KUKA KRL program: EPS_2_251806_BLK210A_A_20260223023028.src

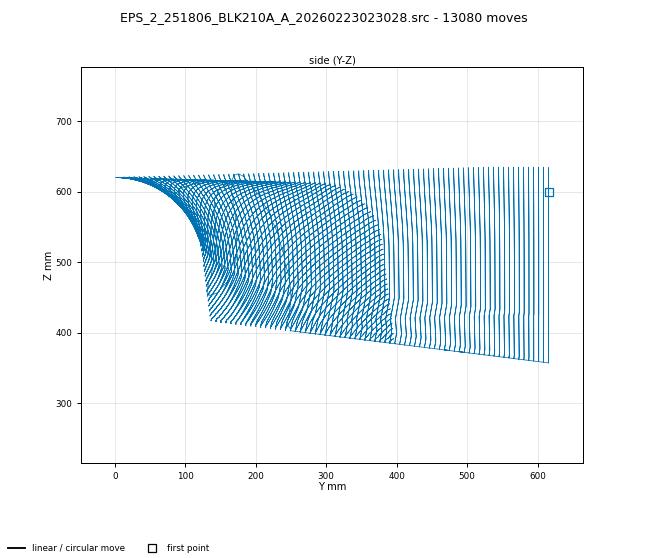
[picture p0: tool path of EPS_2_251806_BLK210A_A_20260223023028.src, 13080 of 13082 moves have a stored position in this frame; points joined in program order, loops and branches not executed]
&ACCESS RVP
&REL 4
&COMMENT QRS 19112012
&PARAM EDITMASK = *
DEF PART()
EXT BAS (BAS_COMMAND :IN,REAL :IN )
INT I
BAS (#INITMOV,0 )

;KUKA QRS Post kuka4.cps  Date:22-06-2017 !

File_ID=3078

QRS_PRE_INIT()

;Init var - Until changes are made in qrs_pre_init
Outlet_Square_prg=0
Inlet_1_Square_prg=0
Inlet_2_Square_prg=0
Inlet_3_Square_prg=0
Inlet_4_Square_prg=0
Inlet_5_Square_prg=0

Outlet_1={X 0.000, Y 530.070, Z 534.500, B 0.000, E1 0.000 }
Inlet_1={X 0.000, Y 550.980, Z 509.500, B 0.000, E1 180.000 }
Outlet_1_type=201
Inlet_1_type=0
;QRS#1=Sidecore dimensions
;QRS#2=200-8" PVC SDR 35
;QRS#3=DeadEnd 201
;QRS#4=
;QRS#5=
;QRS#6=
;QRS#7=
;QRS#8=
;QRS#9=12-08 PSX
;QRS#10=

;QRS#11=
;QRS#12=
;QRS#13=
;QRS#14=
;QRS#15=
;QRS#16=1220x127x914 3'
;QRS#17=EPS Height
;QRS#18=635
;QRS#19=*
;QRS#20= UPDATED VERSION 22-06-2017
;QRS#21=*
Outlet_Square=0100
Inlet_1_Square=00
Inlet_2_Square=0
Inlet_3_Square=0
Inlet_4_Square=0
Inlet_5_Square=0
Mill_Square=1
Outlet_Square_Prg=204
Inlet_1_Square_prg=0

QRS_INIT()

$ADVANCE=5

; T1
PTP {E1 173.602,E2 173.602}
PTP {X 0,Y 615.507,A -85,B 0,C 180,E1 173.602,E2 173.602,E3 0,E4 0,E5 0,E6 0}
QRS_SPEED_INIT()
LIN {X 0,Y 615.507,Z 600,A -85,B 0,C 180,E1 173.602,E2 173.602,E3 0,E4 0,E5 0,E6 0} C_VEL
LIN {X 0,Y 615.507,Z 367.362,A -85,B 0,C 180,E1 173.602,E2 173.602} C_VEL
LIN {X 0,Y 615.507,Z 359.181,A -85,B 0,C 180,E1 173.602,E2 173.602} C_VEL
LIN {X 0,Y 615.49,Z 357.181,A -85,B 0,C 180,E1 173.415,E2 173.415} C_VEL
LIN {X 0,Y 615.478,Z 357.192,A -85,B 0,C 180,E1 170.801,E2 170.801} C_VEL
LIN {X 0,Y 615.484,Z 357.193,A -85,B 0,C 180,E1 168.14,E2 168.14} C_VEL
LIN {X 0,Y 615.49,Z 357.182,A -85,B 0,C 180,E1 165.451,E2 165.451} C_VEL
LIN {X 0,Y 615.489,Z 357.193,A -85,B 0,C 180,E1 162.73,E2 162.73} C_VEL
LIN {X 0,Y 615.483,Z 357.188,A -85,B 0,C 180,E1 159.968,E2 159.968} C_VEL
LIN {X 0,Y 615.491,Z 357.182,A -85,B 0,C 180,E1 157.652,E2 157.652} C_VEL
LIN {X 0,Y 615.477,Z 357.19,A -85,B 0,C 180,E1 155.008,E2 155.008} C_VEL
LIN {X 0,Y 615.482,Z 357.194,A -85,B 0,C 180,E1 152.823,E2 152.823} C_VEL
LIN {X 0,Y 615.482,Z 357.192,A -85,B 0,C 180,E1 150.205,E2 150.205} C_VEL
LIN {X 0,Y 615.489,Z 357.182,A -85,B 0,C 180,E1 147.543,E2 147.543} C_VEL
LIN {X 0,Y 615.477,Z 357.188,A -85,B 0,C 180,E1 145.185,E2 145.185} C_VEL
LIN {X 0,Y 615.491,Z 357.197,A -85,B 0,C 180,E1 142.759,E2 142.759} C_VEL
LIN {X 0,Y 615.487,Z 357.184,A -85,B 0,C 180,E1 139.91,E2 139.91} C_VEL
LIN {X 0,Y 615.493,Z 357.181,A -85,B 0,C 180,E1 137.648,E2 137.648} C_VEL
LIN {X 0,Y 615.481,Z 357.195,A -85,B 0,C 180,E1 134.932,E2 134.932} C_VEL
LIN {X 0,Y 615.482,Z 357.186,A -85,B 0,C 180,E1 132.08,E2 132.08} C_VEL
LIN {X 0,Y 615.494,Z 357.181,A -85,B 0,C 180,E1 129.749,E2 129.749} C_VEL
LIN {X 0,Y 615.483,Z 357.196,A -85,B 0,C 180,E1 126.937,E2 126.937} C_VEL
LIN {X 0,Y 615.492,Z 357.2,A -85,B 0,C 180,E1 124.702,E2 124.702} C_VEL
LIN {X 0,Y 615.48,Z 357.191,A -85,B 0,C 180,E1 122.33,E2 122.33} C_VEL
LIN {X 0,Y 615.497,Z 357.18,A -85,B 0,C 180,E1 119.797,E2 119.797} C_VEL
LIN {X 0,Y 615.486,Z 357.195,A -85,B 0,C 180,E1 117.046,E2 117.046} C_VEL
LIN {X 0,Y 615.479,Z 357.188,A -85,B 0,C 180,E1 114.272,E2 114.272} C_VEL
LIN {X 0,Y 615.477,Z 357.188,A -85,B 0,C 180,E1 111.432,E2 111.432} C_VEL
LIN {X 0,Y 615.482,Z 357.195,A -85,B 0,C 180,E1 108.605,E2 108.605} C_VEL
LIN {X 0,Y 615.486,Z 357.182,A -85,B 0,C 180,E1 105.905,E2 105.905} C_VEL
LIN {X 0,Y 615.48,Z 357.194,A -85,B 0,C 180,E1 103.201,E2 103.201} C_VEL
LIN {X 0,Y 615.479,Z 357.192,A -85,B 0,C 180,E1 100.527,E2 100.527} C_VEL
LIN {X 0,Y 615.488,Z 357.182,A -85,B 0,C 180,E1 97.876,E2 97.876} C_VEL
LIN {X 0,Y 615.482,Z 357.194,A -85,B 0,C 180,E1 95.241,E2 95.241} C_VEL
LIN {X 0,Y 615.477,Z 357.193,A -85,B 0,C 180,E1 92.618,E2 92.618} C_VEL
LIN {X 0,Y 615.486,Z 357.182,A -85,B 0,C 180,E1 90,E2 90} C_VEL
LIN {X 0,Y 615.477,Z 357.193,A -85,B 0,C 180,E1 87.382,E2 87.382} C_VEL
LIN {X 0,Y 615.482,Z 357.194,A -85,B 0,C 180,E1 84.759,E2 84.759} C_VEL
LIN {X 0,Y 615.488,Z 357.182,A -85,B 0,C 180,E1 82.125,E2 82.125} C_VEL
LIN {X 0,Y 615.479,Z 357.192,A -85,B 0,C 180,E1 79.473,E2 79.473} C_VEL
LIN {X 0,Y 615.48,Z 357.194,A -85,B 0,C 180,E1 76.799,E2 76.799} C_VEL
LIN {X 0,Y 615.486,Z 357.182,A -85,B 0,C 180,E1 74.095,E2 74.095} C_VEL
LIN {X 0,Y 615.484,Z 357.196,A -85,B 0,C 180,E1 71.354,E2 71.354} C_VEL
LIN {X 0,Y 615.477,Z 357.188,A -85,B 0,C 180,E1 68.568,E2 68.568} C_VEL
LIN {X 0,Y 615.486,Z 357.183,A -85,B 0,C 180,E1 65.991,E2 65.991} C_VEL
LIN {X 0,Y 615.48,Z 357.192,A -85,B 0,C 180,E1 63.556,E2 63.556} C_VEL
LIN {X 0,Y 615.49,Z 357.197,A -85,B 0,C 180,E1 61.343,E2 61.343} C_VEL
LIN {X 0,Y 615.482,Z 357.193,A -85,B 0,C 180,E1 58.914,E2 58.914} C_VEL
LIN {X 0,Y 615.482,Z 357.184,A -85,B 0,C 180,E1 56.466,E2 56.466} C_VEL
LIN {X 0,Y 615.489,Z 357.182,A -85,B 0,C 180,E1 54.165,E2 54.165} C_VEL
LIN {X 0,Y 615.483,Z 357.185,A -85,B 0,C 180,E1 51.932,E2 51.932} C_VEL
LIN {X 0,Y 615.485,Z 357.2,A -85,B 0,C 180,E1 49.394,E2 49.394} C_VEL
LIN {X 0,Y 615.476,Z 357.189,A -85,B 0,C 180,E1 46.755,E2 46.755} C_VEL
LIN {X 0,Y 615.484,Z 357.185,A -85,B 0,C 180,E1 43.998,E2 43.998} C_VEL
LIN {X 0,Y 615.488,Z 357.198,A -85,B 0,C 180,E1 41.473,E2 41.473} C_VEL
LIN {X 0,Y 615.476,Z 357.191,A -85,B 0,C 180,E1 38.905,E2 38.905} C_VEL
LIN {X 0,Y 615.488,Z 357.182,A -85,B 0,C 180,E1 36.424,E2 36.424} C_VEL
LIN {X 0,Y 615.487,Z 357.198,A -85,B 0,C 180,E1 33.535,E2 33.535} C_VEL
LIN {X 0,Y 615.478,Z 357.189,A -85,B 0,C 180,E1 30.92,E2 30.92} C_VEL
LIN {X 0,Y 615.491,Z 357.181,A -85,B 0,C 180,E1 28.453,E2 28.453} C_VEL
LIN {X 0,Y 615.489,Z 357.198,A -85,B 0,C 180,E1 25.571,E2 25.571} C_VEL
LIN {X 0,Y 615.476,Z 357.187,A -85,B 0,C 180,E1 22.845,E2 22.845} C_VEL
LIN {X 0,Y 615.486,Z 357.182,A -85,B 0,C 180,E1 20.559,E2 20.559} C_VEL
LIN {X 0,Y 615.482,Z 357.19,A -85,B 0,C 180,E1 17.957,E2 17.957} C_VEL
LIN {X 0,Y 615.486,Z 357.192,A -85,B 0,C 180,E1 15.226,E2 15.226} C_VEL
LIN {X 0,Y 615.485,Z 357.183,A -85,B 0,C 180,E1 12.53,E2 12.53} C_VEL
LIN {X 0,Y 615.481,Z 357.194,A -85,B 0,C 180,E1 9.862,E2 9.862} C_VEL
LIN {X 0,Y 615.483,Z 357.191,A -85,B 0,C 180,E1 7.215,E2 7.215} C_VEL
LIN {X 0,Y 615.491,Z 357.181,A -85,B 0,C 180,E1 4.584,E2 4.584} C_VEL
LIN {X 0,Y 615.484,Z 357.192,A -85,B 0,C 180,E1 1.963,E2 1.963} C_VEL
LIN {X 0,Y 615.484,Z 357.193,A -85,B 0,C 180,E1 -0.655,E2 -0.655} C_VEL
LIN {X 0,Y 615.485,Z 357.183,A -85,B 0,C 180,E1 -3.273,E2 -3.273} C_VEL
LIN {X 0,Y 615.484,Z 357.19,A -85,B 0,C 180,E1 -5.899,E2 -5.899} C_VEL
LIN {X 0,Y 615.489,Z 357.194,A -85,B 0,C 180,E1 -8.537,E2 -8.537} C_VEL
LIN {X 0,Y 615.483,Z 357.183,A -85,B 0,C 180,E1 -11.194,E2 -11.194} C_VEL
LIN {X 0,Y 615.485,Z 357.192,A -85,B 0,C 180,E1 -13.935,E2 -13.935} C_VEL
LIN {X 0,Y 615.481,Z 357.192,A -85,B 0,C 180,E1 -16.587,E2 -16.587} C_VEL
LIN {X 0,Y 615.486,Z 357.183,A -85,B 0,C 180,E1 -19.338,E2 -19.338} C_VEL
LIN {X 0,Y 615.493,Z 357.2,A -85,B 0,C 180,E1 -22.137,E2 -22.137} C_VEL
LIN {X 0,Y 615.476,Z 357.185,A -85,B 0,C 180,E1 -24.993,E2 -24.993} C_VEL
LIN {X 0,Y 615.481,Z 357.184,A -85,B 0,C 180,E1 -27.178,E2 -27.178} C_VEL
LIN {X 0,Y 615.485,Z 357.192,A -85,B 0,C 180,E1 -29.796,E2 -29.796} C_VEL
LIN {X 0,Y 615.489,Z 357.191,A -85,B 0,C 180,E1 -32.458,E2 -32.458} C_VEL
LIN {X 0,Y 615.477,Z 357.186,A -85,B 0,C 180,E1 -34.816,E2 -34.816} C_VEL
LIN {X 0,Y 615.489,Z 357.182,A -85,B 0,C 180,E1 -37.242,E2 -37.242} C_VEL
LIN {X 0,Y 615.498,Z 357.2,A -85,B 0,C 180,E1 -40.091,E2 -40.091} C_VEL
LIN {X 0,Y 615.493,Z 357.191,A -85,B 0,C 180,E1 -42.353,E2 -42.353} C_VEL
LIN {X 0,Y 615.481,Z 357.184,A -85,B 0,C 180,E1 -45.07,E2 -45.07} C_VEL
LIN {X 0,Y 615.489,Z 357.199,A -85,B 0,C 180,E1 -47.92,E2 -47.92} C_VEL
LIN {X 0,Y 615.495,Z 357.192,A -85,B 0,C 180,E1 -50.251,E2 -50.251} C_VEL
LIN {X 0,Y 615.483,Z 357.183,A -85,B 0,C 180,E1 -53.064,E2 -53.064} C_VEL
LIN {X 0,Y 615.496,Z 357.2,A -85,B 0,C 180,E1 -55.979,E2 -55.979} C_VEL
LIN {X 0,Y 615.482,Z 357.183,A -85,B 0,C 180,E1 -58.915,E2 -58.915} C_VEL
LIN {X 0,Y 615.486,Z 357.191,A -85,B 0,C 180,E1 -61.551,E2 -61.551} C_VEL
LIN {X 0,Y 615.481,Z 357.188,A -85,B 0,C 180,E1 -64.433,E2 -64.433} C_VEL
LIN {X 0,Y 615.497,Z 357.361,A -85,B 0,C 180,E1 -65.958,E2 -65.958} C_VEL
LIN {X 0,Y 615.496,Z 372.441,A -85,B 0,C 180,E1 -68.569,E2 -68.569} C_VEL
LIN {X 0,Y 615.482,Z 389.222,A -85,B 0,C 180,E1 -71.398,E2 -71.398} C_VEL
LIN {X 0,Y 615.49,Z 405.467,A -85,B 0,C 180,E1 -74.095,E2 -74.095} C_VEL
LIN {X 0,Y 615.497,Z 422.987,A -85,B 0,C 180,E1 -76.967,E2 -76.967} C_VEL
LIN {X 0,Y 615.495,Z 424.551,A -85,B 0,C 180,E1 -77.135,E2 -77.135} C_VEL
LIN {X 0,Y 615.497,Z 530.847,A -85,B 0,C 180,E1 -78.411,E2 -78.411} C_VEL
LIN {X 0,Y 615.499,Z 543.354,A -85,B 0,C 180,E1 -78.682,E2 -78.682} C_VEL
LIN {X 0,Y 615.496,Z 556.502,A -85,B 0,C 180,E1 -79.109,E2 -79.109} C_VEL
LIN {X 0,Y 615.484,Z 568.484,A -85,B 0,C 180,E1 -79.64,E2 -79.64} C_VEL
LIN {X 0,Y 615.487,Z 580,A -85,B 0,C 180,E1 -80.304,E2 -80.304} C_VEL
LIN {X 0,Y 615.499,Z 590.345,A -85,B 0,C 180,E1 -81.05,E2 -81.05} C_VEL
LIN {X 0,Y 615.497,Z 598.815,A -85,B 0,C 180,E1 -81.794,E2 -81.794} C_VEL
LIN {X 0,Y 615.498,Z 606.609,A -85,B 0,C 180,E1 -82.62,E2 -82.62} C_VEL
LIN {X 0,Y 615.496,Z 614.205,A -85,B 0,C 180,E1 -83.608,E2 -83.608} C_VEL
LIN {X 0,Y 615.498,Z 621.206,A -85,B 0,C 180,E1 -84.759,E2 -84.759} C_VEL
LIN {X 0,Y 615.493,Z 625.853,A -85,B 0,C 180,E1 -85.744,E2 -85.744} C_VEL
LIN {X 0,Y 615.495,Z 629.399,A -85,B 0,C 180,E1 -86.727,E2 -86.727} C_VEL
LIN {X 0,Y 615.497,Z 631.233,A -85,B 0,C 180,E1 -87.382,E2 -87.382} C_VEL
LIN {X 0,Y 615.497,Z 632.608,A -85,B 0,C 180,E1 -88.037,E2 -88.037} C_VEL
LIN {X 0,Y 615.496,Z 634.174,A -85,B 0,C 180,E1 -89.346,E2 -89.346} C_VEL
LIN {X 0,Y 615.494,Z 634.389,A -85,B 0,C 180,E1 -90,E2 -90} C_VEL
LIN {X 0,Y 615.496,Z 633.58,A -85,B 0,C 180,E1 -91.309,E2 -91.309} C_VEL
LIN {X 0,Y 615.497,Z 632.608,A -85,B 0,C 180,E1 -91.963,E2 -91.963} C_VEL
LIN {X 0,Y 615.497,Z 631.232,A -85,B 0,C 180,E1 -92.618,E2 -92.618} C_VEL
LIN {X 0,Y 615.496,Z 628.349,A -85,B 0,C 180,E1 -93.601,E2 -93.601} C_VEL
LIN {X 0,Y 615.498,Z 624.441,A -85,B 0,C 180,E1 -94.585,E2 -94.585} C_VEL
LIN {X 0,Y 615.499,Z 619.404,A -85,B 0,C 180,E1 -95.57,E2 -95.57} C_VEL
LIN {X 0,Y 615.497,Z 612.87,A -85,B 0,C 180,E1 -96.583,E2 -96.583} C_VEL
LIN {X 0,Y 615.497,Z 605.132,A -85,B 0,C 180,E1 -97.545,E2 -97.545} C_VEL
LIN {X 0,Y 615.498,Z 597.044,A -85,B 0,C 180,E1 -98.371,E2 -98.371} C_VEL
LIN {X 0,Y 615.499,Z 587.166,A -85,B 0,C 180,E1 -99.199,E2 -99.199} C_VEL
LIN {X 0,Y 615.488,Z 575.98,A -85,B 0,C 180,E1 -99.945,E2 -99.945} C_VEL
LIN {X 0,Y 615.486,Z 565.021,A -85,B 0,C 180,E1 -100.527,E2 -100.527} C_VEL
LIN {X 0,Y 615.499,Z 552.418,A -85,B 0,C 180,E1 -101.042,E2 -101.042} C_VEL
LIN {X 0,Y 615.499,Z 540.06,A -85,B 0,C 180,E1 -101.401,E2 -101.401} C_VEL
LIN {X 0,Y 615.498,Z 526.459,A -85,B 0,C 180,E1 -101.652,E2 -101.652} C_VEL
LIN {X 0,Y 615.495,Z 424.541,A -85,B 0,C 180,E1 -102.865,E2 -102.865} C_VEL
LIN {X 0,Y 615.497,Z 422.984,A -85,B 0,C 180,E1 -103.033,E2 -103.033} C_VEL
LIN {X 0,Y 615.49,Z 405.464,A -85,B 0,C 180,E1 -105.905,E2 -105.905} C_VEL
LIN {X 0,Y 615.484,Z 388.96,A -85,B 0,C 180,E1 -108.646,E2 -108.646} C_VEL
LIN {X 0,Y 615.496,Z 372.438,A -85,B 0,C 180,E1 -111.432,E2 -111.432} C_VEL
LIN {X 0,Y 615.497,Z 357.361,A -85,B 0,C 180,E1 -114.042,E2 -114.042} C_VEL
LIN {X 0,Y 615.485,Z 357.192,A -85,B 0,C 180,E1 -116.444,E2 -116.444} C_VEL
LIN {X 0,Y 615.489,Z 357.186,A -85,B 0,C 180,E1 -118.658,E2 -118.658} C_VEL
LIN {X 0,Y 615.482,Z 357.183,A -85,B 0,C 180,E1 -121.085,E2 -121.085} C_VEL
LIN {X 0,Y 615.498,Z 357.199,A -85,B 0,C 180,E1 -124.021,E2 -124.021} C_VEL
LIN {X 0,Y 615.483,Z 357.183,A -85,B 0,C 180,E1 -126.936,E2 -126.936} C_VEL
LIN {X 0,Y 615.495,Z 357.192,A -85,B 0,C 180,E1 -129.749,E2 -129.749} C_VEL
LIN {X 0,Y 615.485,Z 357.191,A -85,B 0,C 180,E1 -132.353,E2 -132.353} C_VEL
LIN {X 0,Y 615.479,Z 357.184,A -85,B 0,C 180,E1 -135.069,E2 -135.069} C_VEL
LIN {X 0,Y 615.496,Z 357.2,A -85,B 0,C 180,E1 -137.918,E2 -137.918} C_VEL
LIN {X 0,Y 615.486,Z 357.192,A -85,B 0,C 180,E1 -140.249,E2 -140.249} C_VEL
LIN {X 0,Y 615.478,Z 357.185,A -85,B 0,C 180,E1 -143.064,E2 -143.064} C_VEL
LIN {X 0,Y 615.495,Z 357.198,A -85,B 0,C 180,E1 -145.978,E2 -145.978} C_VEL
LIN {X 0,Y 615.485,Z 357.189,A -85,B 0,C 180,E1 -148.314,E2 -148.314} C_VEL
LIN {X 0,Y 615.488,Z 357.183,A -85,B 0,C 180,E1 -150.593,E2 -150.593} C_VEL
LIN {X 0,Y 615.481,Z 357.184,A -85,B 0,C 180,E1 -152.955,E2 -152.955} C_VEL
LIN {X 0,Y 615.496,Z 357.197,A -85,B 0,C 180,E1 -155.728,E2 -155.728} C_VEL
LIN {X 0,Y 615.495,Z 357.182,A -85,B 0,C 180,E1 -158.568,E2 -158.568} C_VEL
LIN {X 0,Y 615.485,Z 357.191,A -85,B 0,C 180,E1 -161.395,E2 -161.395} C_VEL
LIN {X 0,Y 615.483,Z 357.193,A -85,B 0,C 180,E1 -164.094,E2 -164.094} C_VEL
LIN {X 0,Y 615.484,Z 357.183,A -85,B 0,C 180,E1 -166.798,E2 -166.798} C_VEL
LIN {X 0,Y 615.493,Z 357.193,A -85,B 0,C 180,E1 -169.473,E2 -169.473} C_VEL
LIN {X 0,Y 615.482,Z 357.19,A -85,B 0,C 180,E1 -172.124,E2 -172.124} C_VEL
LIN {X 0,Y 615.484,Z 357.183,A -85,B 0,C 180,E1 -174.758,E2 -174.758} C_VEL
LIN {X 0,Y 615.489,Z 357.192,A -85,B 0,C 180,E1 -177.382,E2 -177.382} C_VEL
LIN {X 0,Y 615.484,Z 357.192,A -85,B 0,C 180,E1 -180,E2 -180} C_VEL
LIN {X 0,Y 615.49,Z 357.182,A -85,B 0,C 180,E1 -182.617,E2 -182.617} C_VEL
LIN {X 0,Y 615.484,Z 357.191,A -85,B 0,C 180,E1 -185.241,E2 -185.241} C_VEL
LIN {X 0,Y 615.49,Z 357.181,A -85,B 0,C 180,E1 -186.585,E2 -186.585} C_VEL
LIN {X 0,Y 614.809,Z 357.338,A -85,B 0,C 180,E1 -187.131,E2 -187.131} C_VEL
LIN {X 0,Y 611.968,Z 357.753,A -85,B 0,C 180,E1 -188.017,E2 -188.017} C_VEL
LIN {X 0,Y 609.575,Z 358.065,A -85,B 0,C 180,E1 -188.729,E2 -188.729} C_VEL
LIN {X 0,Y 608.541,Z 358.183,A -85,B 0,C 180,E1 -189.279,E2 -189.279} C_VEL
LIN {X 0,Y 608.453,Z 358.191,A -85,B 0,C 180,E1 -189.465,E2 -189.465} C_VEL
LIN {X 0,Y 608.46,Z 358.19,A -85,B 0,C 180,E1 -191.999,E2 -191.999} C_VEL
LIN {X 0,Y 608.477,Z 358.185,A -85,B 0,C 180,E1 -194.72,E2 -194.72} C_VEL
LIN {X 0,Y 608.453,Z 358.197,A -85,B 0,C 180,E1 -197.476,E2 -197.476} C_VEL
LIN {X 0,Y 608.461,Z 358.186,A -85,B 0,C 180,E1 -200.274,E2 -200.274} C_VEL
LIN {X 0,Y 608.455,Z 358.187,A -85,B 0,C 180,E1 -202.476,E2 -202.476} C_VEL
LIN {X 0,Y 608.451,Z 358.187,A -85,B 0,C 180,E1 -204.571,E2 -204.571} C_VEL
LIN {X 0,Y 608.474,Z 358.191,A -85,B 0,C 180,E1 -207.207,E2 -207.207} C_VEL
LIN {X 0,Y 608.465,Z 358.188,A -85,B 0,C 180,E1 -209.972,E2 -209.972} C_VEL
LIN {X 0,Y 608.463,Z 358.186,A -85,B 0,C 180,E1 -212.523,E2 -212.523} C_VEL
LIN {X 0,Y 608.44,Z 358.197,A -85,B 0,C 180,E1 -215.277,E2 -215.277} C_VEL
LIN {X 0,Y 608.469,Z 358.19,A -85,B 0,C 180,E1 -217.746,E2 -217.746} C_VEL
LIN {X 0,Y 608.449,Z 358.187,A -85,B 0,C 180,E1 -220.329,E2 -220.329} C_VEL
LIN {X 0,Y 608.483,Z 358.194,A -85,B 0,C 180,E1 -223.311,E2 -223.311} C_VEL
LIN {X 0,Y 608.468,Z 358.185,A -85,B 0,C 180,E1 -226.131,E2 -226.131} C_VEL
LIN {X 0,Y 608.449,Z 358.19,A -85,B 0,C 180,E1 -228.823,E2 -228.823} C_VEL
LIN {X 0,Y 608.468,Z 358.194,A -85,B 0,C 180,E1 -231.412,E2 -231.412} C_VEL
LIN {X 0,Y 608.475,Z 358.185,A -85,B 0,C 180,E1 -233.95,E2 -233.95} C_VEL
LIN {X 0,Y 608.46,Z 358.186,A -85,B 0,C 180,E1 -236.329,E2 -236.329} C_VEL
LIN {X 0,Y 608.474,Z 358.187,A -85,B 0,C 180,E1 -238.727,E2 -238.727} C_VEL
LIN {X 0,Y 608.473,Z 358.192,A -85,B 0,C 180,E1 -241.379,E2 -241.379} C_VEL
LIN {X 0,Y 608.47,Z 358.185,A -85,B 0,C 180,E1 -244.278,E2 -244.278} C_VEL
LIN {X 0,Y 608.449,Z 358.193,A -85,B 0,C 180,E1 -246.876,E2 -246.876} C_VEL
LIN {X 0,Y 608.46,Z 358.188,A -85,B 0,C 180,E1 -249.726,E2 -249.726} C_VEL
LIN {X 0,Y 608.45,Z 358.189,A -85,B 0,C 180,E1 -252.523,E2 -252.523} C_VEL
LIN {X 0,Y 608.469,Z 358.193,A -85,B 0,C 180,E1 -255.279,E2 -255.279} C_VEL
LIN {X 0,Y 608.461,Z 358.186,A -85,B 0,C 180,E1 -258,E2 -258} C_VEL
LIN {X 0,Y 608.466,Z 358.19,A -85,B 0,C 180,E1 -260.694,E2 -260.694} C_VEL
LIN {X 0,Y 608.475,Z 358.19,A -85,B 0,C 180,E1 -263.367,E2 -263.367} C_VEL
LIN {X 0,Y 608.455,Z 358.187,A -85,B 0,C 180,E1 -266.026,E2 -266.026} C_VEL
LIN {X 0,Y 608.465,Z 358.191,A -85,B 0,C 180,E1 -268.676,E2 -268.676} C_VEL
LIN {X 0,Y 608.465,Z 358.191,A -85,B 0,C 180,E1 -271.323,E2 -271.323} C_VEL
LIN {X 0,Y 608.456,Z 358.187,A -85,B 0,C 180,E1 -273.974,E2 -273.974} C_VEL
LIN {X 0,Y 608.474,Z 358.19,A -85,B 0,C 180,E1 -276.632,E2 -276.632} C_VEL
LIN {X 0,Y 608.466,Z 358.19,A -85,B 0,C 180,E1 -279.306,E2 -279.306} C_VEL
LIN {X 0,Y 608.461,Z 358.186,A -85,B 0,C 180,E1 -281.999,E2 -281.999} C_VEL
LIN {X 0,Y 608.469,Z 358.193,A -85,B 0,C 180,E1 -284.72,E2 -284.72} C_VEL
LIN {X 0,Y 608.45,Z 358.189,A -85,B 0,C 180,E1 -287.476,E2 -287.476} C_VEL
LIN {X 0,Y 608.46,Z 358.188,A -85,B 0,C 180,E1 -290.274,E2 -290.274} C_VEL
LIN {X 0,Y 608.449,Z 358.193,A -85,B 0,C 180,E1 -293.124,E2 -293.124} C_VEL
LIN {X 0,Y 608.47,Z 358.185,A -85,B 0,C 180,E1 -295.722,E2 -295.722} C_VEL
LIN {X 0,Y 608.472,Z 358.192,A -85,B 0,C 180,E1 -298.621,E2 -298.621} C_VEL
LIN {X 0,Y 608.472,Z 358.187,A -85,B 0,C 180,E1 -301.316,E2 -301.316} C_VEL
LIN {X 0,Y 608.469,Z 358.185,A -85,B 0,C 180,E1 -303.735,E2 -303.735} C_VEL
LIN {X 0,Y 608.473,Z 358.186,A -85,B 0,C 180,E1 -306.09,E2 -306.09} C_VEL
LIN {X 0,Y 608.468,Z 358.194,A -85,B 0,C 180,E1 -308.587,E2 -308.587} C_VEL
LIN {X 0,Y 608.456,Z 358.187,A -85,B 0,C 180,E1 -311.342,E2 -311.342} C_VEL
LIN {X 0,Y 608.45,Z 358.191,A -85,B 0,C 180,E1 -314.264,E2 -314.264} C_VEL
LIN {X 0,Y 608.452,Z 358.192,A -85,B 0,C 180,E1 -317.041,E2 -317.041} C_VEL
LIN {X 0,Y 608.45,Z 358.187,A -85,B 0,C 180,E1 -319.697,E2 -319.697} C_VEL
LIN {X 0,Y 608.469,Z 358.19,A -85,B 0,C 180,E1 -322.254,E2 -322.254} C_VEL
LIN {X 0,Y 608.469,Z 358.188,A -85,B 0,C 180,E1 -325.09,E2 -325.09} C_VEL
LIN {X 0,Y 608.471,Z 358.186,A -85,B 0,C 180,E1 -327.906,E2 -327.906} C_VEL
LIN {X 0,Y 608.467,Z 358.19,A -85,B 0,C 180,E1 -330.221,E2 -330.221} C_VEL
LIN {X 0,Y 608.474,Z 358.191,A -85,B 0,C 180,E1 -332.792,E2 -332.792} C_VEL
LIN {X 0,Y 608.451,Z 358.187,A -85,B 0,C 180,E1 -335.429,E2 -335.429} C_VEL
LIN {X 0,Y 608.475,Z 358.192,A -85,B 0,C 180,E1 -338.309,E2 -338.309} C_VEL
LIN {X 0,Y 608.466,Z 358.186,A -85,B 0,C 180,E1 -341.283,E2 -341.283} C_VEL
LIN {X 0,Y 608.46,Z 358.188,A -85,B 0,C 180,E1 -343.907,E2 -343.907} C_VEL
LIN {X 0,Y 608.461,Z 358.193,A -85,B 0,C 180,E1 -346.644,E2 -346.644} C_VEL
LIN {X 0,Y 608.465,Z 358.185,A -85,B 0,C 180,E1 -349.351,E2 -349.351} C_VEL
LIN {X 0,Y 608.476,Z 358.188,A -85,B 0,C 180,E1 -352.033,E2 -352.033} C_VEL
LIN {X 0,Y 608.463,Z 358.191,A -85,B 0,C 180,E1 -354.699,E2 -354.699} C_VEL
LIN {X 0,Y 608.48,Z 358.184,A -85,B 0,C 180,E1 -357.352,E2 -357.352} C_VEL
LIN {X 0,Y 608.472,Z 358.189,A -85,B 0,C 180,E1 -360,E2 -360} C_VEL
LIN {X 0,Y 608.48,Z 358.189,A -85,B 0,C 180,E1 -362.648,E2 -362.648} C_VEL
LIN {X 0,Y 608.463,Z 358.186,A -85,B 0,C 180,E1 -365.302,E2 -365.302} C_VEL
LIN {X 0,Y 608.474,Z 358.189,A -85,B 0,C 180,E1 -367.967,E2 -367.967} C_VEL
LIN {X 0,Y 608.463,Z 358.187,A -85,B 0,C 180,E1 -370.957,E2 -370.957} C_VEL
LIN {X 0,Y 608.461,Z 358.186,A -85,B 0,C 180,E1 -373.357,E2 -373.357} C_VEL
LIN {X 0,Y 608.46,Z 358.194,A -85,B 0,C 180,E1 -376.094,E2 -376.094} C_VEL
LIN {X 0,Y 608.452,Z 358.188,A -85,B 0,C 180,E1 -378.87,E2 -378.87} C_VEL
LIN {X 0,Y 608.476,Z 358.187,A -85,B 0,C 180,E1 -381.692,E2 -381.692} C_VEL
LIN {X 0,Y 608.452,Z 358.191,A -85,B 0,C 180,E1 -384.571,E2 -384.571} C_VEL
LIN {X 0,Y 608.473,Z 358.184,A -85,B 0,C 180,E1 -387.208,E2 -387.208} C_VEL
LIN {X 0,Y 608.47,Z 358.193,A -85,B 0,C 180,E1 -389.974,E2 -389.974} C_VEL
LIN {X 0,Y 608.463,Z 358.19,A -85,B 0,C 180,E1 -392.524,E2 -392.524} C_VEL
LIN {X 0,Y 608.439,Z 358.189,A -85,B 0,C 180,E1 -395.278,E2 -395.278} C_VEL
LIN {X 0,Y 608.473,Z 358.19,A -85,B 0,C 180,E1 -397.746,E2 -397.746} C_VEL
LIN {X 0,Y 608.454,Z 358.193,A -85,B 0,C 180,E1 -400.33,E2 -400.33} C_VEL
LIN {X 0,Y 608.453,Z 358.187,A -85,B 0,C 180,E1 -402.96,E2 -402.96} C_VEL
LIN {X 0,Y 608.457,Z 358.192,A -85,B 0,C 180,E1 -405.736,E2 -405.736} C_VEL
LIN {X 0,Y 608.457,Z 358.188,A -85,B 0,C 180,E1 -408.659,E2 -408.659} C_VEL
LIN {X 0,Y 608.471,Z 358.187,A -85,B 0,C 180,E1 -411.413,E2 -411.413} C_VEL
LIN {X 0,Y 608.479,Z 358.195,A -85,B 0,C 180,E1 -413.951,E2 -413.951} C_VEL
LIN {X 0,Y 608.464,Z 358.19,A -85,B 0,C 180,E1 -416.33,E2 -416.33} C_VEL
LIN {X 0,Y 608.46,Z 358.187,A -85,B 0,C 180,E1 -418.731,E2 -418.731} C_VEL
LIN {X 0,Y 608.474,Z 358.187,A -85,B 0,C 180,E1 -421.38,E2 -421.38} C_VEL
LIN {X 0,Y 608.471,Z 358.19,A -85,B 0,C 180,E1 -424.28,E2 -424.28} C_VEL
LIN {X 0,Y 608.491,Z 358.355,A -85,B 0,C 180,E1 -425.845,E2 -425.845} C_VEL
LIN {X 0,Y 608.547,Z 372.465,A -85,B 0,C 180,E1 -428.312,E2 -428.312} C_VEL
LIN {X 0,Y 608.511,Z 389.856,A -85,B 0,C 180,E1 -431.274,E2 -431.274} C_VEL
LIN {X 0,Y 608.496,Z 406.613,A -85,B 0,C 180,E1 -434.08,E2 -434.08} C_VEL
LIN {X 0,Y 608.473,Z 424.032,A -85,B 0,C 180,E1 -436.942,E2 -436.942} C_VEL
LIN {X 0,Y 608.582,Z 425.271,A -85,B 0,C 180,E1 -437.008,E2 -437.008} C_VEL
LIN {X 0,Y 608.549,Z 530.958,A -85,B 0,C 180,E1 -438.277,E2 -438.277} C_VEL
LIN {X 0,Y 608.547,Z 544.234,A -85,B 0,C 180,E1 -438.572,E2 -438.572} C_VEL
LIN {X 0,Y 608.54,Z 557.395,A -85,B 0,C 180,E1 -439.011,E2 -439.011} C_VEL
LIN {X 0,Y 608.507,Z 568.632,A -85,B 0,C 180,E1 -439.52,E2 -439.52} C_VEL
LIN {X 0,Y 608.48,Z 580.198,A -85,B 0,C 180,E1 -440.191,E2 -440.191} C_VEL
LIN {X 0,Y 608.485,Z 590.596,A -85,B 0,C 180,E1 -440.946,E2 -440.946} C_VEL
LIN {X 0,Y 608.475,Z 599.115,A -85,B 0,C 180,E1 -441.699,E2 -441.699} C_VEL
LIN {X 0,Y 608.471,Z 606.963,A -85,B 0,C 180,E1 -442.534,E2 -442.534} C_VEL
LIN {X 0,Y 608.46,Z 614.287,A -85,B 0,C 180,E1 -443.485,E2 -443.485} C_VEL
LIN {X 0,Y 608.45,Z 619.866,A -85,B 0,C 180,E1 -444.366,E2 -444.366} C_VEL
LIN {X 0,Y 608.432,Z 624.949,A -85,B 0,C 180,E1 -445.362,E2 -445.362} C_VEL
LIN {X 0,Y 608.449,Z 628.895,A -85,B 0,C 180,E1 -446.358,E2 -446.358} C_VEL
LIN {X 0,Y 608.425,Z 631.809,A -85,B 0,C 180,E1 -447.352,E2 -447.352} C_VEL
LIN {X 0,Y 608.443,Z 633.202,A -85,B 0,C 180,E1 -448.014,E2 -448.014} C_VEL
LIN {X 0,Y 608.439,Z 634.784,A -85,B 0,C 180,E1 -449.338,E2 -449.338} C_VEL
LIN {X 0,Y 608.434,Z 635,A -85,B 0,C 180,E1 -450,E2 -450} C_VEL
LIN {X 0,Y 608.448,Z 634.183,A -85,B 0,C 180,E1 -451.324,E2 -451.324} C_VEL
LIN {X 0,Y 608.443,Z 633.201,A -85,B 0,C 180,E1 -451.986,E2 -451.986} C_VEL
LIN {X 0,Y 608.425,Z 631.808,A -85,B 0,C 180,E1 -452.648,E2 -452.648} C_VEL
LIN {X 0,Y 608.449,Z 628.894,A -85,B 0,C 180,E1 -453.643,E2 -453.643} C_VEL
LIN {X 0,Y 608.432,Z 624.948,A -85,B 0,C 180,E1 -454.638,E2 -454.638} C_VEL
LIN {X 0,Y 608.437,Z 618.877,A -85,B 0,C 180,E1 -455.801,E2 -455.801} C_VEL
LIN {X 0,Y 608.462,Z 612.234,A -85,B 0,C 180,E1 -456.799,E2 -456.799} C_VEL
LIN {X 0,Y 608.456,Z 603.988,A -85,B 0,C 180,E1 -457.8,E2 -457.8} C_VEL
LIN {X 0,Y 608.472,Z 595.532,A -85,B 0,C 180,E1 -458.636,E2 -458.636} C_VEL
LIN {X 0,Y 608.472,Z 585.09,A -85,B 0,C 180,E1 -459.474,E2 -459.474} C_VEL
LIN {X 0,Y 608.495,Z 574.756,A -85,B 0,C 180,E1 -460.145,E2 -460.145} C_VEL
LIN {X 0,Y 608.522,Z 563.235,A -85,B 0,C 180,E1 -460.741,E2 -460.741} C_VEL
LIN {X 0,Y 608.533,Z 551.861,A -85,B 0,C 180,E1 -461.193,E2 -461.193} C_VEL
LIN {X 0,Y 608.551,Z 539.26,A -85,B 0,C 180,E1 -461.554,E2 -461.554} C_VEL
LIN {X 0,Y 608.574,Z 526.597,A -85,B 0,C 180,E1 -461.786,E2 -461.786} C_VEL
LIN {X 0,Y 608.533,Z 424.577,A -85,B 0,C 180,E1 -463.015,E2 -463.015} C_VEL
LIN {X 0,Y 608.492,Z 423.167,A -85,B 0,C 180,E1 -463.186,E2 -463.186} C_VEL
LIN {X 0,Y 608.488,Z 405.575,A -85,B 0,C 180,E1 -466.093,E2 -466.093} C_VEL
LIN {X 0,Y 608.513,Z 389.019,A -85,B 0,C 180,E1 -468.868,E2 -468.868} C_VEL
LIN {X 0,Y 608.547,Z 372.462,A -85,B 0,C 180,E1 -471.689,E2 -471.689} C_VEL
LIN {X 0,Y 608.491,Z 358.344,A -85,B 0,C 180,E1 -474.155,E2 -474.155} C_VEL
LIN {X 0,Y 608.449,Z 358.189,A -85,B 0,C 180,E1 -476.774,E2 -476.774} C_VEL
LIN {X 0,Y 608.469,Z 358.185,A -85,B 0,C 180,E1 -479.02,E2 -479.02} C_VEL
LIN {X 0,Y 608.448,Z 358.189,A -85,B 0,C 180,E1 -481.317,E2 -481.317} C_VEL
LIN {X 0,Y 608.473,Z 358.19,A -85,B 0,C 180,E1 -483.735,E2 -483.735} C_VEL
LIN {X 0,Y 608.48,Z 358.194,A -85,B 0,C 180,E1 -486.09,E2 -486.09} C_VEL
LIN {X 0,Y 608.471,Z 358.187,A -85,B 0,C 180,E1 -488.587,E2 -488.587} C_VEL
LIN {X 0,Y 608.457,Z 358.188,A -85,B 0,C 180,E1 -491.341,E2 -491.341} C_VEL
LIN {X 0,Y 608.459,Z 358.192,A -85,B 0,C 180,E1 -494.264,E2 -494.264} C_VEL
LIN {X 0,Y 608.453,Z 358.187,A -85,B 0,C 180,E1 -497.04,E2 -497.04} C_VEL
LIN {X 0,Y 608.455,Z 358.193,A -85,B 0,C 180,E1 -499.697,E2 -499.697} C_VEL
LIN {X 0,Y 608.472,Z 358.19,A -85,B 0,C 180,E1 -502.254,E2 -502.254} C_VEL
LIN {X 0,Y 608.439,Z 358.189,A -85,B 0,C 180,E1 -504.722,E2 -504.722} C_VEL
LIN {X 0,Y 608.46,Z 358.19,A -85,B 0,C 180,E1 -507.477,E2 -507.477} C_VEL
LIN {X 0,Y 608.469,Z 358.19,A -85,B 0,C 180,E1 -510.22,E2 -510.22} C_VEL
LIN {X 0,Y 608.477,Z 358.184,A -85,B 0,C 180,E1 -512.792,E2 -512.792} C_VEL
LIN {X 0,Y 608.454,Z 358.191,A -85,B 0,C 180,E1 -515.429,E2 -515.429} C_VEL
LIN {X 0,Y 608.476,Z 358.187,A -85,B 0,C 180,E1 -518.308,E2 -518.308} C_VEL
LIN {X 0,Y 608.469,Z 358.188,A -85,B 0,C 180,E1 -521.283,E2 -521.283} C_VEL
LIN {X 0,Y 608.461,Z 358.194,A -85,B 0,C 180,E1 -523.906,E2 -523.906} C_VEL
LIN {X 0,Y 608.462,Z 358.186,A -85,B 0,C 180,E1 -526.643,E2 -526.643} C_VEL
LIN {X 0,Y 608.466,Z 358.19,A -85,B 0,C 180,E1 -529.35,E2 -529.35} C_VEL
LIN {X 0,Y 608.475,Z 358.189,A -85,B 0,C 180,E1 -532.033,E2 -532.033} C_VEL
LIN {X 0,Y 608.463,Z 358.186,A -85,B 0,C 180,E1 -534.698,E2 -534.698} C_VEL
LIN {X 0,Y 608.48,Z 358.189,A -85,B 0,C 180,E1 -537.352,E2 -537.352} C_VEL
LIN {X 0,Y 608.475,Z 358.189,A -85,B 0,C 180,E1 -540,E2 -540} C_VEL
LIN {X 0,Y 608.48,Z 358.184,A -85,B 0,C 180,E1 -542.648,E2 -542.648} C_VEL
LIN {X 0,Y 608.463,Z 358.191,A -85,B 0,C 180,E1 -545.301,E2 -545.301} C_VEL
LIN {X 0,Y 608.476,Z 358.188,A -85,B 0,C 180,E1 -547.967,E2 -547.967} C_VEL
LIN {X 0,Y 608.453,Z 358.191,A -85,B 0,C 180,E1 -549.465,E2 -549.465} C_VEL
LIN {X 0,Y 607.777,Z 358.275,A -85,B 0,C 180,E1 -550.018,E2 -550.018} C_VEL
LIN {X 0,Y 604.924,Z 358.628,A -85,B 0,C 180,E1 -550.915,E2 -550.915} C_VEL
LIN {X 0,Y 602.521,Z 358.935,A -85,B 0,C 180,E1 -551.636,E2 -551.636} C_VEL
LIN {X 0,Y 601.491,Z 359.056,A -85,B 0,C 180,E1 -552.193,E2 -552.193} C_VEL
LIN {X 0,Y 601.408,Z 359.065,A -85,B 0,C 180,E1 -552.381,E2 -552.381} C_VEL
LIN {X 0,Y 601.43,Z 359.063,A -85,B 0,C 180,E1 -554.896,E2 -554.896} C_VEL
LIN {X 0,Y 601.431,Z 359.064,A -85,B 0,C 180,E1 -556.985,E2 -556.985} C_VEL
LIN {X 0,Y 601.406,Z 359.07,A -85,B 0,C 180,E1 -559.809,E2 -559.809} C_VEL
LIN {X 0,Y 601.408,Z 359.065,A -85,B 0,C 180,E1 -562.683,E2 -562.683} C_VEL
LIN {X 0,Y 601.4,Z 359.068,A -85,B 0,C 180,E1 -564.878,E2 -564.878} C_VEL
LIN {X 0,Y 601.419,Z 359.067,A -85,B 0,C 180,E1 -567.867,E2 -567.867} C_VEL
LIN {X 0,Y 601.424,Z 359.064,A -85,B 0,C 180,E1 -570.164,E2 -570.164} C_VEL
LIN {X 0,Y 601.424,Z 359.064,A -85,B 0,C 180,E1 -572.716,E2 -572.716} C_VEL
LIN {X 0,Y 601.405,Z 359.07,A -85,B 0,C 180,E1 -575.114,E2 -575.114} C_VEL
LIN {X 0,Y 601.432,Z 359.072,A -85,B 0,C 180,E1 -577.419,E2 -577.419} C_VEL
LIN {X 0,Y 601.407,Z 359.066,A -85,B 0,C 180,E1 -579.995,E2 -579.995} C_VEL
LIN {X 0,Y 601.412,Z 359.065,A -85,B 0,C 180,E1 -582.67,E2 -582.67} C_VEL
LIN {X 0,Y 601.421,Z 359.07,A -85,B 0,C 180,E1 -585.482,E2 -585.482} C_VEL
LIN {X 0,Y 601.42,Z 359.062,A -85,B 0,C 180,E1 -588.407,E2 -588.407} C_VEL
LIN {X 0,Y 601.433,Z 359.065,A -85,B 0,C 180,E1 -590.875,E2 -590.875} C_VEL
LIN {X 0,Y 601.441,Z 359.063,A -85,B 0,C 180,E1 -593.734,E2 -593.734} C_VEL
LIN {X 0,Y 601.429,Z 359.062,A -85,B 0,C 180,E1 -596.064,E2 -596.064} C_VEL
LIN {X 0,Y 601.438,Z 359.062,A -85,B 0,C 180,E1 -598.542,E2 -598.542} C_VEL
LIN {X 0,Y 601.432,Z 359.07,A -85,B 0,C 180,E1 -601.373,E2 -601.373} C_VEL
LIN {X 0,Y 601.411,Z 359.065,A -85,B 0,C 180,E1 -604.132,E2 -604.132} C_VEL
LIN {X 0,Y 601.418,Z 359.066,A -85,B 0,C 180,E1 -606.59,E2 -606.59} C_VEL
LIN {X 0,Y 601.429,Z 359.067,A -85,B 0,C 180,E1 -609.478,E2 -609.478} C_VEL
LIN {X 0,Y 601.397,Z 359.067,A -85,B 0,C 180,E1 -612.312,E2 -612.312} C_VEL
LIN {X 0,Y 601.411,Z 359.066,A -85,B 0,C 180,E1 -614.409,E2 -614.409} C_VEL
LIN {X 0,Y 601.415,Z 359.074,A -85,B 0,C 180,E1 -617.172,E2 -617.172} C_VEL
LIN {X 0,Y 601.434,Z 359.062,A -85,B 0,C 180,E1 -619.905,E2 -619.905} C_VEL
LIN {X 0,Y 601.439,Z 359.065,A -85,B 0,C 180,E1 -622.615,E2 -622.615} C_VEL
LIN {X 0,Y 601.416,Z 359.07,A -85,B 0,C 180,E1 -625.308,E2 -625.308} C_VEL
LIN {X 0,Y 601.435,Z 359.062,A -85,B 0,C 180,E1 -627.991,E2 -627.991} C_VEL
LIN {X 0,Y 601.446,Z 359.066,A -85,B 0,C 180,E1 -630.669,E2 -630.669} C_VEL
LIN {X 0,Y 601.426,Z 359.067,A -85,B 0,C 180,E1 -633.349,E2 -633.349} C_VEL
LIN {X 0,Y 601.437,Z 359.061,A -85,B 0,C 180,E1 -636.037,E2 -636.037} C_VEL
LIN {X 0,Y 601.43,Z 359.069,A -85,B 0,C 180,E1 -638.737,E2 -638.737} C_VEL
LIN {X 0,Y 601.432,Z 359.064,A -85,B 0,C 180,E1 -641.458,E2 -641.458} C_VEL
LIN {X 0,Y 601.416,Z 359.065,A -85,B 0,C 180,E1 -644.205,E2 -644.205} C_VEL
LIN {X 0,Y 601.428,Z 359.071,A -85,B 0,C 180,E1 -646.986,E2 -646.986} C_VEL
LIN {X 0,Y 601.402,Z 359.066,A -85,B 0,C 180,E1 -649.809,E2 -649.809} C_VEL
LIN {X 0,Y 601.408,Z 359.073,A -85,B 0,C 180,E1 -652.683,E2 -652.683} C_VEL
LIN {X 0,Y 601.4,Z 359.076,A -85,B 0,C 180,E1 -654.878,E2 -654.878} C_VEL
LIN {X 0,Y 601.417,Z 359.064,A -85,B 0,C 180,E1 -657.867,E2 -657.867} C_VEL
LIN {X 0,Y 601.444,Z 359.061,A -85,B 0,C 180,E1 -660.163,E2 -660.163} C_VEL
LIN {X 0,Y 601.417,Z 359.074,A -85,B 0,C 180,E1 -662.716,E2 -662.716} C_VEL
LIN {X 0,Y 601.417,Z 359.068,A -85,B 0,C 180,E1 -665.116,E2 -665.116} C_VEL
LIN {X 0,Y 601.429,Z 359.063,A -85,B 0,C 180,E1 -667.419,E2 -667.419} C_VEL
LIN {X 0,Y 601.408,Z 359.065,A -85,B 0,C 180,E1 -669.994,E2 -669.994} C_VEL
LIN {X 0,Y 601.406,Z 359.074,A -85,B 0,C 180,E1 -672.67,E2 -672.67} C_VEL
LIN {X 0,Y 601.418,Z 359.064,A -85,B 0,C 180,E1 -675.482,E2 -675.482} C_VEL
LIN {X 0,Y 601.423,Z 359.069,A -85,B 0,C 180,E1 -678.406,E2 -678.406} C_VEL
LIN {X 0,Y 601.429,Z 359.069,A -85,B 0,C 180,E1 -680.875,E2 -680.875} C_VEL
LIN {X 0,Y 601.437,Z 359.061,A -85,B 0,C 180,E1 -683.734,E2 -683.734} C_VEL
LIN {X 0,Y 601.426,Z 359.072,A -85,B 0,C 180,E1 -686.687,E2 -686.687} C_VEL
LIN {X 0,Y 601.425,Z 359.066,A -85,B 0,C 180,E1 -689.059,E2 -689.059} C_VEL
LIN {X 0,Y 601.431,Z 359.062,A -85,B 0,C 180,E1 -691.374,E2 -691.374} C_VEL
LIN {X 0,Y 601.412,Z 359.068,A -85,B 0,C 180,E1 -694.131,E2 -694.131} C_VEL
LIN {X 0,Y 601.416,Z 359.073,A -85,B 0,C 180,E1 -696.59,E2 -696.59} C_VEL
LIN {X 0,Y 601.428,Z 359.062,A -85,B 0,C 180,E1 -699.479,E2 -699.479} C_VEL
LIN {X 0,Y 601.397,Z 359.073,A -85,B 0,C 180,E1 -702.312,E2 -702.312} C_VEL
LIN {X 0,Y 601.414,Z 359.074,A -85,B 0,C 180,E1 -704.409,E2 -704.409} C_VEL
LIN {X 0,Y 601.418,Z 359.064,A -85,B 0,C 180,E1 -707.172,E2 -707.172} C_VEL
LIN {X 0,Y 601.431,Z 359.063,A -85,B 0,C 180,E1 -709.905,E2 -709.905} C_VEL
LIN {X 0,Y 601.448,Z 359.067,A -85,B 0,C 180,E1 -712.615,E2 -712.615} C_VEL
LIN {X 0,Y 601.427,Z 359.062,A -85,B 0,C 180,E1 -715.308,E2 -715.308} C_VEL
LIN {X 0,Y 601.424,Z 359.067,A -85,B 0,C 180,E1 -717.991,E2 -717.991} C_VEL
LIN {X 0,Y 601.449,Z 359.064,A -85,B 0,C 180,E1 -720.67,E2 -720.67} C_VEL
LIN {X 0,Y 601.428,Z 359.062,A -85,B 0,C 180,E1 -723.35,E2 -723.35} C_VEL
LIN {X 0,Y 601.411,Z 359.07,A -85,B 0,C 180,E1 -726.037,E2 -726.037} C_VEL
LIN {X 0,Y 601.435,Z 359.063,A -85,B 0,C 180,E1 -728.738,E2 -728.738} C_VEL
LIN {X 0,Y 601.431,Z 359.062,A -85,B 0,C 180,E1 -731.459,E2 -731.459} C_VEL
LIN {X 0,Y 601.415,Z 359.074,A -85,B 0,C 180,E1 -734.206,E2 -734.206} C_VEL
LIN {X 0,Y 601.429,Z 359.062,A -85,B 0,C 180,E1 -736.986,E2 -736.986} C_VEL
LIN {X 0,Y 601.407,Z 359.068,A -85,B 0,C 180,E1 -739.81,E2 -739.81} C_VEL
LIN {X 0,Y 601.408,Z 359.068,A -85,B 0,C 180,E1 -742.683,E2 -742.683} C_VEL
LIN {X 0,Y 601.4,Z 359.066,A -85,B 0,C 180,E1 -744.879,E2 -744.879} C_VEL
LIN {X 0,Y 601.421,Z 359.068,A -85,B 0,C 180,E1 -747.868,E2 -747.868} C_VEL
LIN {X 0,Y 601.445,Z 359.071,A -85,B 0,C 180,E1 -750.163,E2 -750.163} C_VEL
LIN {X 0,Y 601.424,Z 359.064,A -85,B 0,C 180,E1 -752.717,E2 -752.717} C_VEL
LIN {X 0,Y 601.405,Z 359.065,A -85,B 0,C 180,E1 -755.115,E2 -755.115} C_VEL
LIN {X 0,Y 601.434,Z 359.063,A -85,B 0,C 180,E1 -757.42,E2 -757.42} C_VEL
LIN {X 0,Y 601.412,Z 359.074,A -85,B 0,C 180,E1 -759.995,E2 -759.995} C_VEL
LIN {X 0,Y 601.413,Z 359.066,A -85,B 0,C 180,E1 -762.671,E2 -762.671} C_VEL
LIN {X 0,Y 601.424,Z 359.065,A -85,B 0,C 180,E1 -765.483,E2 -765.483} C_VEL
LIN {X 0,Y 601.422,Z 359.066,A -85,B 0,C 180,E1 -768.407,E2 -768.407} C_VEL
LIN {X 0,Y 601.435,Z 359.061,A -85,B 0,C 180,E1 -770.876,E2 -770.876} C_VEL
LIN {X 0,Y 601.444,Z 359.067,A -85,B 0,C 180,E1 -773.734,E2 -773.734} C_VEL
LIN {X 0,Y 601.434,Z 359.07,A -85,B 0,C 180,E1 -776.065,E2 -776.065} C_VEL
LIN {X 0,Y 601.43,Z 359.064,A -85,B 0,C 180,E1 -778.544,E2 -778.544} C_VEL
LIN {X 0,Y 601.439,Z 359.062,A -85,B 0,C 180,E1 -781.211,E2 -781.211} C_VEL
LIN {X 0,Y 601.404,Z 359.072,A -85,B 0,C 180,E1 -783.637,E2 -783.637} C_VEL
LIN {X 0,Y 601.468,Z 359.234,A -85,B 0,C 180,E1 -785.701,E2 -785.701} C_VEL
LIN {X 0,Y 601.57,Z 368.533,A -85,B 0,C 180,E1 -787.36,E2 -787.36} C_VEL
LIN {X 0,Y 601.558,Z 383.847,A -85,B 0,C 180,E1 -790.018,E2 -790.018} C_VEL
LIN {X 0,Y 601.501,Z 401.439,A -85,B 0,C 180,E1 -793.017,E2 -793.017} C_VEL
LIN {X 0,Y 601.428,Z 418.665,A -85,B 0,C 180,E1 -795.907,E2 -795.907} C_VEL
LIN {X 0,Y 601.462,Z 424.247,A -85,B 0,C 180,E1 -796.808,E2 -796.808} C_VEL
LIN {X 0,Y 601.688,Z 426.75,A -85,B 0,C 180,E1 -796.878,E2 -796.878} C_VEL
LIN {X 0,Y 601.596,Z 530.914,A -85,B 0,C 180,E1 -798.14,E2 -798.14} C_VEL
LIN {X 0,Y 601.59,Z 544.242,A -85,B 0,C 180,E1 -798.439,E2 -798.439} C_VEL
LIN {X 0,Y 601.547,Z 556.667,A -85,B 0,C 180,E1 -798.854,E2 -798.854} C_VEL
LIN {X 0,Y 601.518,Z 568.617,A -85,B 0,C 180,E1 -799.396,E2 -799.396} C_VEL
LIN {X 0,Y 601.481,Z 580.195,A -85,B 0,C 180,E1 -800.076,E2 -800.076} C_VEL
LIN {X 0,Y 601.444,Z 590.595,A -85,B 0,C 180,E1 -800.839,E2 -800.839} C_VEL
LIN {X 0,Y 601.429,Z 599.114,A -85,B 0,C 180,E1 -801.601,E2 -801.601} C_VEL
LIN {X 0,Y 601.418,Z 606.963,A -85,B 0,C 180,E1 -802.446,E2 -802.446} C_VEL
LIN {X 0,Y 601.37,Z 614.223,A -85,B 0,C 180,E1 -803.398,E2 -803.398} C_VEL
LIN {X 0,Y 601.373,Z 619.863,A -85,B 0,C 180,E1 -804.299,E2 -804.299} C_VEL
LIN {X 0,Y 601.336,Z 624.943,A -85,B 0,C 180,E1 -805.308,E2 -805.308} C_VEL
LIN {X 0,Y 601.367,Z 628.888,A -85,B 0,C 180,E1 -806.315,E2 -806.315} C_VEL
LIN {X 0,Y 601.325,Z 631.805,A -85,B 0,C 180,E1 -807.321,E2 -807.321} C_VEL
LIN {X 0,Y 601.341,Z 633.203,A -85,B 0,C 180,E1 -807.991,E2 -807.991} C_VEL
LIN {X 0,Y 601.339,Z 634.784,A -85,B 0,C 180,E1 -809.331,E2 -809.331} C_VEL
LIN {X 0,Y 601.335,Z 635,A -85,B 0,C 180,E1 -810,E2 -810} C_VEL
LIN {X 0,Y 601.348,Z 634.183,A -85,B 0,C 180,E1 -811.34,E2 -811.34} C_VEL
LIN {X 0,Y 601.341,Z 633.203,A -85,B 0,C 180,E1 -812.009,E2 -812.009} C_VEL
LIN {X 0,Y 601.325,Z 631.804,A -85,B 0,C 180,E1 -812.68,E2 -812.68} C_VEL
LIN {X 0,Y 601.367,Z 628.887,A -85,B 0,C 180,E1 -813.685,E2 -813.685} C_VEL
LIN {X 0,Y 601.336,Z 624.942,A -85,B 0,C 180,E1 -814.693,E2 -814.693} C_VEL
LIN {X 0,Y 601.372,Z 619.861,A -85,B 0,C 180,E1 -815.701,E2 -815.701} C_VEL
LIN {X 0,Y 601.382,Z 613.472,A -85,B 0,C 180,E1 -816.711,E2 -816.711} C_VEL
LIN {X 0,Y 601.396,Z 605.477,A -85,B 0,C 180,E1 -817.723,E2 -817.723} C_VEL
LIN {X 0,Y 601.423,Z 597.334,A -85,B 0,C 180,E1 -818.569,E2 -818.569} C_VEL
LIN {X 0,Y 601.449,Z 587.381,A -85,B 0,C 180,E1 -819.415,E2 -819.415} C_VEL
LIN {X 0,Y 601.494,Z 576.172,A -85,B 0,C 180,E1 -820.179,E2 -820.179} C_VEL
LIN {X 0,Y 601.538,Z 563.906,A -85,B 0,C 180,E1 -820.836,E2 -820.836} C_VEL
LIN {X 0,Y 601.566,Z 551.349,A -85,B 0,C 180,E1 -821.34,E2 -821.34} C_VEL
LIN {X 0,Y 601.607,Z 538.34,A -85,B 0,C 180,E1 -821.711,E2 -821.711} C_VEL
LIN {X 0,Y 601.624,Z 525.08,A -85,B 0,C 180,E1 -821.946,E2 -821.946} C_VEL
LIN {X 0,Y 601.549,Z 425.225,A -85,B 0,C 180,E1 -823.147,E2 -823.147} C_VEL
LIN {X 0,Y 601.472,Z 424.027,A -85,B 0,C 180,E1 -823.214,E2 -823.214} C_VEL
LIN {X 0,Y 601.465,Z 406.61,A -85,B 0,C 180,E1 -826.112,E2 -826.112} C_VEL
LIN {X 0,Y 601.525,Z 390.464,A -85,B 0,C 180,E1 -828.848,E2 -828.848} C_VEL
LIN {X 0,Y 601.574,Z 373.497,A -85,B 0,C 180,E1 -831.773,E2 -831.773} C_VEL
LIN {X 0,Y 601.592,Z 360.045,A -85,B 0,C 180,E1 -834.134,E2 -834.134} C_VEL
LIN {X 0,Y 601.448,Z 359.174,A -85,B 0,C 180,E1 -834.341,E2 -834.341} C_VEL
LIN {X 0,Y 601.449,Z 359.06,A -85,B 0,C 180,E1 -837.111,E2 -837.111} C_VEL
LIN {X 0,Y 601.452,Z 359.069,A -85,B 0,C 180,E1 -840.162,E2 -840.162} C_VEL
LIN {X 0,Y 601.422,Z 359.064,A -85,B 0,C 180,E1 -842.715,E2 -842.715} C_VEL
LIN {X 0,Y 601.418,Z 359.064,A -85,B 0,C 180,E1 -845.114,E2 -845.114} C_VEL
LIN {X 0,Y 601.436,Z 359.063,A -85,B 0,C 180,E1 -847.419,E2 -847.419} C_VEL
LIN {X 0,Y 601.414,Z 359.074,A -85,B 0,C 180,E1 -849.994,E2 -849.994} C_VEL
LIN {X 0,Y 601.411,Z 359.066,A -85,B 0,C 180,E1 -852.67,E2 -852.67} C_VEL
LIN {X 0,Y 601.427,Z 359.065,A -85,B 0,C 180,E1 -855.482,E2 -855.482} C_VEL
LIN {X 0,Y 601.427,Z 359.066,A -85,B 0,C 180,E1 -858.406,E2 -858.406} C_VEL
LIN {X 0,Y 601.434,Z 359.061,A -85,B 0,C 180,E1 -860.875,E2 -860.875} C_VEL
LIN {X 0,Y 601.443,Z 359.068,A -85,B 0,C 180,E1 -863.734,E2 -863.734} C_VEL
LIN {X 0,Y 601.429,Z 359.062,A -85,B 0,C 180,E1 -866.686,E2 -866.686} C_VEL
LIN {X 0,Y 601.431,Z 359.062,A -85,B 0,C 180,E1 -869.058,E2 -869.058} C_VEL
LIN {X 0,Y 601.432,Z 359.065,A -85,B 0,C 180,E1 -871.373,E2 -871.373} C_VEL
LIN {X 0,Y 601.404,Z 359.071,A -85,B 0,C 180,E1 -873.636,E2 -873.636} C_VEL
LIN {X 0,Y 601.419,Z 359.064,A -85,B 0,C 180,E1 -876.589,E2 -876.589} C_VEL
LIN {X 0,Y 601.431,Z 359.067,A -85,B 0,C 180,E1 -879.478,E2 -879.478} C_VEL
LIN {X 0,Y 601.397,Z 359.068,A -85,B 0,C 180,E1 -882.311,E2 -882.311} C_VEL
LIN {X 0,Y 601.414,Z 359.065,A -85,B 0,C 180,E1 -884.408,E2 -884.408} C_VEL
LIN {X 0,Y 601.42,Z 359.065,A -85,B 0,C 180,E1 -887.171,E2 -887.171} C_VEL
LIN {X 0,Y 601.433,Z 359.068,A -85,B 0,C 180,E1 -889.905,E2 -889.905} C_VEL
LIN {X 0,Y 601.438,Z 359.061,A -85,B 0,C 180,E1 -892.614,E2 -892.614} C_VEL
LIN {X 0,Y 601.424,Z 359.067,A -85,B 0,C 180,E1 -895.308,E2 -895.308} C_VEL
LIN {X 0,Y 601.424,Z 359.067,A -85,B 0,C 180,E1 -897.991,E2 -897.991} C_VEL
LIN {X 0,Y 601.45,Z 359.058,A -85,B 0,C 180,E1 -900.669,E2 -900.669} C_VEL
LIN {X 0,Y 601.429,Z 359.068,A -85,B 0,C 180,E1 -903.349,E2 -903.349} C_VEL
LIN {X 0,Y 601.41,Z 359.068,A -85,B 0,C 180,E1 -906.037,E2 -906.037} C_VEL
LIN {X 0,Y 601.434,Z 359.061,A -85,B 0,C 180,E1 -908.737,E2 -908.737} C_VEL
LIN {X 0,Y 601.432,Z 359.07,A -85,B 0,C 180,E1 -911.458,E2 -911.458} C_VEL
LIN {X 0,Y 601.408,Z 359.065,A -85,B 0,C 180,E1 -912.381,E2 -912.381} C_VEL
LIN {X 0,Y 600.743,Z 359.15,A -85,B 0,C 180,E1 -912.941,E2 -912.941} C_VEL
LIN {X 0,Y 597.894,Z 359.508,A -85,B 0,C 180,E1 -913.848,E2 -913.848} C_VEL
LIN {X 0,Y 595.484,Z 359.807,A -85,B 0,C 180,E1 -914.579,E2 -914.579} C_VEL
LIN {X 0,Y 594.447,Z 359.936,A -85,B 0,C 180,E1 -915.142,E2 -915.142} C_VEL
LIN {X 0,Y 594.361,Z 359.946,A -85,B 0,C 180,E1 -915.333,E2 -915.333} C_VEL
LIN {X 0,Y 594.353,Z 359.946,A -85,B 0,C 180,E1 -917.905,E2 -917.905} C_VEL
LIN {X 0,Y 594.401,Z 359.938,A -85,B 0,C 180,E1 -920.775,E2 -920.775} C_VEL
LIN {X 0,Y 594.387,Z 359.946,A -85,B 0,C 180,E1 -923.704,E2 -923.704} C_VEL
LIN {X 0,Y 594.383,Z 359.94,A -85,B 0,C 180,E1 -926.699,E2 -926.699} C_VEL
LIN {X 0,Y 594.378,Z 359.943,A -85,B 0,C 180,E1 -928.998,E2 -928.998} C_VEL
LIN {X 0,Y 594.39,Z 359.946,A -85,B 0,C 180,E1 -931.645,E2 -931.645} C_VEL
LIN {X 0,Y 594.388,Z 359.938,A -85,B 0,C 180,E1 -934.579,E2 -934.579} C_VEL
LIN {X 0,Y 594.382,Z 359.945,A -85,B 0,C 180,E1 -937.086,E2 -937.086} C_VEL
LIN {X 0,Y 594.37,Z 359.945,A -85,B 0,C 180,E1 -939.774,E2 -939.774} C_VEL
LIN {X 0,Y 594.369,Z 359.942,A -85,B 0,C 180,E1 -942.375,E2 -942.375} C_VEL
LIN {X 0,Y 594.359,Z 359.951,A -85,B 0,C 180,E1 -945.191,E2 -945.191} C_VEL
LIN {X 0,Y 594.379,Z 359.938,A -85,B 0,C 180,E1 -948.151,E2 -948.151} C_VEL
LIN {X 0,Y 594.384,Z 359.949,A -85,B 0,C 180,E1 -951.195,E2 -951.195} C_VEL
LIN {X 0,Y 594.393,Z 359.941,A -85,B 0,C 180,E1 -953.759,E2 -953.759} C_VEL
LIN {X 0,Y 594.375,Z 359.94,A -85,B 0,C 180,E1 -956.239,E2 -956.239} C_VEL
LIN {X 0,Y 594.387,Z 359.942,A -85,B 0,C 180,E1 -958.651,E2 -958.651} C_VEL
LIN {X 0,Y 594.382,Z 359.947,A -85,B 0,C 180,E1 -961.041,E2 -961.041} C_VEL
LIN {X 0,Y 594.385,Z 359.94,A -85,B 0,C 180,E1 -963.976,E2 -963.976} C_VEL
LIN {X 0,Y 594.387,Z 359.94,A -85,B 0,C 180,E1 -966.296,E2 -966.296} C_VEL
LIN {X 0,Y 594.402,Z 359.947,A -85,B 0,C 180,E1 -969.224,E2 -969.224} C_VEL
LIN {X 0,Y 594.379,Z 359.941,A -85,B 0,C 180,E1 -972.096,E2 -972.096} C_VEL
LIN {X 0,Y 594.364,Z 359.943,A -85,B 0,C 180,E1 -974.219,E2 -974.219} C_VEL
LIN {X 0,Y 594.363,Z 359.952,A -85,B 0,C 180,E1 -977.017,E2 -977.017} C_VEL
LIN {X 0,Y 594.393,Z 359.94,A -85,B 0,C 180,E1 -979.784,E2 -979.784} C_VEL
LIN {X 0,Y 594.392,Z 359.942,A -85,B 0,C 180,E1 -982.527,E2 -982.527} C_VEL
LIN {X 0,Y 594.386,Z 359.947,A -85,B 0,C 180,E1 -985.252,E2 -985.252} C_VEL
LIN {X 0,Y 594.404,Z 359.938,A -85,B 0,C 180,E1 -987.967,E2 -987.967} C_VEL
LIN {X 0,Y 594.417,Z 359.941,A -85,B 0,C 180,E1 -990.677,E2 -990.677} C_VEL
LIN {X 0,Y 594.378,Z 359.945,A -85,B 0,C 180,E1 -993.389,E2 -993.389} C_VEL
LIN {X 0,Y 594.39,Z 359.94,A -85,B 0,C 180,E1 -996.108,E2 -996.108} C_VEL
LIN {X 0,Y 594.393,Z 359.948,A -85,B 0,C 180,E1 -998.842,E2 -998.842} C_VEL
LIN {X 0,Y 594.391,Z 359.94,A -85,B 0,C 180,E1 -1001.595,E2 -1001.595} C_VEL
LIN {X 0,Y 594.386,Z 359.943,A -85,B 0,C 180,E1 -1004.377,E2 -1004.377} C_VEL
LIN {X 0,Y 594.386,Z 359.945,A -85,B 0,C 180,E1 -1007.193,E2 -1007.193} C_VEL
LIN {X 0,Y 594.372,Z 359.942,A -85,B 0,C 180,E1 -1010.053,E2 -1010.053} C_VEL
LIN {X 0,Y 594.361,Z 359.951,A -85,B 0,C 180,E1 -1012.967,E2 -1012.967} C_VEL
LIN {X 0,Y 594.373,Z 359.946,A -85,B 0,C 180,E1 -1015.193,E2 -1015.193} C_VEL
LIN {X 0,Y 594.38,Z 359.941,A -85,B 0,C 180,E1 -1017.526,E2 -1017.526} C_VEL
LIN {X 0,Y 594.396,Z 359.941,A -85,B 0,C 180,E1 -1020.331,E2 -1020.331} C_VEL
LIN {X 0,Y 594.373,Z 359.948,A -85,B 0,C 180,E1 -1022.95,E2 -1022.95} C_VEL
LIN {X 0,Y 594.381,Z 359.941,A -85,B 0,C 180,E1 -1025.406,E2 -1025.406} C_VEL
LIN {X 0,Y 594.383,Z 359.941,A -85,B 0,C 180,E1 -1027.94,E2 -1027.94} C_VEL
LIN {X 0,Y 594.374,Z 359.947,A -85,B 0,C 180,E1 -1030.822,E2 -1030.822} C_VEL
LIN {X 0,Y 594.375,Z 359.94,A -85,B 0,C 180,E1 -1033.841,E2 -1033.841} C_VEL
LIN {X 0,Y 594.38,Z 359.95,A -85,B 0,C 180,E1 -1036.702,E2 -1036.702} C_VEL
LIN {X 0,Y 594.368,Z 359.942,A -85,B 0,C 180,E1 -1039.434,E2 -1039.434} C_VEL
LIN {X 0,Y 594.385,Z 359.946,A -85,B 0,C 180,E1 -1042.391,E2 -1042.391} C_VEL
LIN {X 0,Y 594.377,Z 359.949,A -85,B 0,C 180,E1 -1044.672,E2 -1044.672} C_VEL
LIN {X 0,Y 594.374,Z 359.944,A -85,B 0,C 180,E1 -1047.088,E2 -1047.088} C_VEL
LIN {X 0,Y 594.393,Z 359.939,A -85,B 0,C 180,E1 -1049.669,E2 -1049.669} C_VEL
LIN {X 0,Y 594.366,Z 359.951,A -85,B 0,C 180,E1 -1052.539,E2 -1052.539} C_VEL
LIN {X 0,Y 594.373,Z 359.947,A -85,B 0,C 180,E1 -1054.807,E2 -1054.807} C_VEL
LIN {X 0,Y 594.359,Z 359.944,A -85,B 0,C 180,E1 -1057.264,E2 -1057.264} C_VEL
LIN {X 0,Y 594.373,Z 359.942,A -85,B 0,C 180,E1 -1059.947,E2 -1059.947} C_VEL
LIN {X 0,Y 594.386,Z 359.944,A -85,B 0,C 180,E1 -1062.807,E2 -1062.807} C_VEL
LIN {X 0,Y 594.382,Z 359.942,A -85,B 0,C 180,E1 -1065.826,E2 -1065.826} C_VEL
LIN {X 0,Y 594.389,Z 359.949,A -85,B 0,C 180,E1 -1068.405,E2 -1068.405} C_VEL
LIN {X 0,Y 594.394,Z 359.938,A -85,B 0,C 180,E1 -1071.158,E2 -1071.158} C_VEL
LIN {X 0,Y 594.365,Z 359.945,A -85,B 0,C 180,E1 -1073.891,E2 -1073.891} C_VEL
LIN {X 0,Y 594.381,Z 359.946,A -85,B 0,C 180,E1 -1076.611,E2 -1076.611} C_VEL
LIN {X 0,Y 594.418,Z 359.933,A -85,B 0,C 180,E1 -1079.323,E2 -1079.323} C_VEL
LIN {X 0,Y 594.394,Z 359.943,A -85,B 0,C 180,E1 -1082.033,E2 -1082.033} C_VEL
LIN {X 0,Y 594.395,Z 359.942,A -85,B 0,C 180,E1 -1084.748,E2 -1084.748} C_VEL
LIN {X 0,Y 594.397,Z 359.938,A -85,B 0,C 180,E1 -1087.473,E2 -1087.473} C_VEL
LIN {X 0,Y 594.392,Z 359.946,A -85,B 0,C 180,E1 -1090.216,E2 -1090.216} C_VEL
LIN {X 0,Y 594.367,Z 359.943,A -85,B 0,C 180,E1 -1092.983,E2 -1092.983} C_VEL
LIN {X 0,Y 594.367,Z 359.945,A -85,B 0,C 180,E1 -1095.781,E2 -1095.781} C_VEL
LIN {X 0,Y 594.383,Z 359.942,A -85,B 0,C 180,E1 -1098.618,E2 -1098.618} C_VEL
LIN {X 0,Y 594.368,Z 359.942,A -85,B 0,C 180,E1 -1101.504,E2 -1101.504} C_VEL
LIN {X 0,Y 594.385,Z 359.945,A -85,B 0,C 180,E1 -1104.447,E2 -1104.447} C_VEL
LIN {X 0,Y 594.383,Z 359.941,A -85,B 0,C 180,E1 -1106.7,E2 -1106.7} C_VEL
LIN {X 0,Y 594.378,Z 359.941,A -85,B 0,C 180,E1 -1108.999,E2 -1108.999} C_VEL
LIN {X 0,Y 594.391,Z 359.942,A -85,B 0,C 180,E1 -1111.646,E2 -1111.646} C_VEL
LIN {X 0,Y 594.389,Z 359.942,A -85,B 0,C 180,E1 -1114.58,E2 -1114.58} C_VEL
LIN {X 0,Y 594.383,Z 359.94,A -85,B 0,C 180,E1 -1117.087,E2 -1117.087} C_VEL
LIN {X 0,Y 594.374,Z 359.946,A -85,B 0,C 180,E1 -1119.775,E2 -1119.775} C_VEL
LIN {X 0,Y 594.371,Z 359.946,A -85,B 0,C 180,E1 -1122.376,E2 -1122.376} C_VEL
LIN {X 0,Y 594.361,Z 359.943,A -85,B 0,C 180,E1 -1125.192,E2 -1125.192} C_VEL
LIN {X 0,Y 594.383,Z 359.947,A -85,B 0,C 180,E1 -1128.152,E2 -1128.152} C_VEL
LIN {X 0,Y 594.387,Z 359.94,A -85,B 0,C 180,E1 -1131.196,E2 -1131.196} C_VEL
LIN {X 0,Y 594.396,Z 359.945,A -85,B 0,C 180,E1 -1133.759,E2 -1133.759} C_VEL
LIN {X 0,Y 594.38,Z 359.946,A -85,B 0,C 180,E1 -1136.24,E2 -1136.24} C_VEL
LIN {X 0,Y 594.38,Z 359.942,A -85,B 0,C 180,E1 -1138.651,E2 -1138.651} C_VEL
LIN {X 0,Y 594.385,Z 359.941,A -85,B 0,C 180,E1 -1141.043,E2 -1141.043} C_VEL
LIN {X 0,Y 594.388,Z 359.95,A -85,B 0,C 180,E1 -1143.978,E2 -1143.978} C_VEL
LIN {X 0,Y 594.422,Z 360.14,A -85,B 0,C 180,E1 -1145.56,E2 -1145.56} C_VEL
LIN {X 0,Y 594.651,Z 365.221,A -85,B 0,C 180,E1 -1146.492,E2 -1146.492} C_VEL
LIN {X 0,Y 594.562,Z 380.743,A -85,B 0,C 180,E1 -1149.231,E2 -1149.231} C_VEL
LIN {X 0,Y 594.512,Z 397.3,A -85,B 0,C 180,E1 -1152.1,E2 -1152.1} C_VEL
LIN {X 0,Y 594.44,Z 413.856,A -85,B 0,C 180,E1 -1154.924,E2 -1154.924} C_VEL
LIN {X 0,Y 594.422,Z 424.241,A -85,B 0,C 180,E1 -1156.649,E2 -1156.649} C_VEL
LIN {X 0,Y 594.768,Z 426.75,A -85,B 0,C 180,E1 -1156.722,E2 -1156.722} C_VEL
LIN {X 0,Y 594.664,Z 530.86,A -85,B 0,C 180,E1 -1157.999,E2 -1157.999} C_VEL
LIN {X 0,Y 594.638,Z 544.249,A -85,B 0,C 180,E1 -1158.301,E2 -1158.301} C_VEL
LIN {X 0,Y 594.593,Z 557.357,A -85,B 0,C 180,E1 -1158.749,E2 -1158.749} C_VEL
LIN {X 0,Y 594.536,Z 568.602,A -85,B 0,C 180,E1 -1159.27,E2 -1159.27} C_VEL
LIN {X 0,Y 594.467,Z 580.191,A -85,B 0,C 180,E1 -1159.958,E2 -1159.958} C_VEL
LIN {X 0,Y 594.413,Z 590.593,A -85,B 0,C 180,E1 -1160.73,E2 -1160.73} C_VEL
LIN {X 0,Y 594.372,Z 600.792,A -85,B 0,C 180,E1 -1161.672,E2 -1161.672} C_VEL
LIN {X 0,Y 594.316,Z 609.689,A -85,B 0,C 180,E1 -1162.697,E2 -1162.697} C_VEL
LIN {X 0,Y 594.281,Z 616.161,A -85,B 0,C 180,E1 -1163.615,E2 -1163.615} C_VEL
LIN {X 0,Y 594.289,Z 621.67,A -85,B 0,C 180,E1 -1164.572,E2 -1164.572} C_VEL
LIN {X 0,Y 594.27,Z 626.358,A -85,B 0,C 180,E1 -1165.592,E2 -1165.592} C_VEL
LIN {X 0,Y 594.267,Z 629.948,A -85,B 0,C 180,E1 -1166.61,E2 -1166.61} C_VEL
LIN {X 0,Y 594.226,Z 631.798,A -85,B 0,C 180,E1 -1167.289,E2 -1167.289} C_VEL
LIN {X 0,Y 594.24,Z 633.205,A -85,B 0,C 180,E1 -1167.967,E2 -1167.967} C_VEL
LIN {X 0,Y 594.239,Z 634.785,A -85,B 0,C 180,E1 -1169.323,E2 -1169.323} C_VEL
LIN {X 0,Y 594.236,Z 635,A -85,B 0,C 180,E1 -1170,E2 -1170} C_VEL
LIN {X 0,Y 594.247,Z 634.182,A -85,B 0,C 180,E1 -1171.356,E2 -1171.356} C_VEL
LIN {X 0,Y 594.24,Z 633.204,A -85,B 0,C 180,E1 -1172.033,E2 -1172.033} C_VEL
LIN {X 0,Y 594.226,Z 631.797,A -85,B 0,C 180,E1 -1172.712,E2 -1172.712} C_VEL
LIN {X 0,Y 594.288,Z 628.88,A -85,B 0,C 180,E1 -1173.729,E2 -1173.729} C_VEL
LIN {X 0,Y 594.241,Z 624.936,A -85,B 0,C 180,E1 -1174.749,E2 -1174.749} C_VEL
LIN {X 0,Y 594.298,Z 619.858,A -85,B 0,C 180,E1 -1175.769,E2 -1175.769} C_VEL
LIN {X 0,Y 594.316,Z 613.473,A -85,B 0,C 180,E1 -1176.791,E2 -1176.791} C_VEL
LIN {X 0,Y 594.346,Z 605.477,A -85,B 0,C 180,E1 -1177.816,E2 -1177.816} C_VEL
LIN {X 0,Y 594.377,Z 597.334,A -85,B 0,C 180,E1 -1178.671,E2 -1178.671} C_VEL
LIN {X 0,Y 594.411,Z 587.368,A -85,B 0,C 180,E1 -1179.528,E2 -1179.528} C_VEL
LIN {X 0,Y 594.468,Z 576.176,A -85,B 0,C 180,E1 -1180.301,E2 -1180.301} C_VEL
LIN {X 0,Y 594.56,Z 563.709,A -85,B 0,C 180,E1 -1180.974,E2 -1180.974} C_VEL
LIN {X 0,Y 594.6,Z 551.648,A -85,B 0,C 180,E1 -1181.464,E2 -1181.464} C_VEL
LIN {X 0,Y 594.664,Z 539.248,A -85,B 0,C 180,E1 -1181.828,E2 -1181.828} C_VEL
LIN {X 0,Y 594.693,Z 526.597,A -85,B 0,C 180,E1 -1182.065,E2 -1182.065} C_VEL
LIN {X 0,Y 594.662,Z 426.169,A -85,B 0,C 180,E1 -1183.287,E2 -1183.287} C_VEL
LIN {X 0,Y 594.423,Z 424.238,A -85,B 0,C 180,E1 -1183.351,E2 -1183.351} C_VEL
LIN {X 0,Y 594.455,Z 407.645,A -85,B 0,C 180,E1 -1186.131,E2 -1186.131} C_VEL
LIN {X 0,Y 594.541,Z 390.358,A -85,B 0,C 180,E1 -1189.097,E2 -1189.097} C_VEL
LIN {X 0,Y 594.617,Z 373.497,A -85,B 0,C 180,E1 -1192.041,E2 -1192.041} C_VEL
LIN {X 0,Y 594.599,Z 361.101,A -85,B 0,C 180,E1 -1194.247,E2 -1194.247} C_VEL
LIN {X 0,Y 594.392,Z 360.034,A -85,B 0,C 180,E1 -1194.492,E2 -1194.492} C_VEL
LIN {X 0,Y 594.386,Z 359.943,A -85,B 0,C 180,E1 -1196.699,E2 -1196.699} C_VEL
LIN {X 0,Y 594.384,Z 359.941,A -85,B 0,C 180,E1 -1198.998,E2 -1198.998} C_VEL
LIN {X 0,Y 594.38,Z 359.945,A -85,B 0,C 180,E1 -1201.642,E2 -1201.642} C_VEL
LIN {X 0,Y 594.4,Z 359.94,A -85,B 0,C 180,E1 -1204.578,E2 -1204.578} C_VEL
LIN {X 0,Y 594.386,Z 359.939,A -85,B 0,C 180,E1 -1207.086,E2 -1207.086} C_VEL
LIN {X 0,Y 594.378,Z 359.947,A -85,B 0,C 180,E1 -1209.774,E2 -1209.774} C_VEL
LIN {X 0,Y 594.369,Z 359.946,A -85,B 0,C 180,E1 -1212.375,E2 -1212.375} C_VEL
LIN {X 0,Y 594.364,Z 359.943,A -85,B 0,C 180,E1 -1215.191,E2 -1215.191} C_VEL
LIN {X 0,Y 594.372,Z 359.946,A -85,B 0,C 180,E1 -1217.625,E2 -1217.625} C_VEL
LIN {X 0,Y 594.392,Z 359.943,A -85,B 0,C 180,E1 -1220.32,E2 -1220.32} C_VEL
LIN {X 0,Y 594.385,Z 359.94,A -85,B 0,C 180,E1 -1222.913,E2 -1222.913} C_VEL
LIN {X 0,Y 594.382,Z 359.95,A -85,B 0,C 180,E1 -1225.861,E2 -1225.861} C_VEL
LIN {X 0,Y 594.39,Z 359.94,A -85,B 0,C 180,E1 -1228.651,E2 -1228.651} C_VEL
LIN {X 0,Y 594.383,Z 359.94,A -85,B 0,C 180,E1 -1231.041,E2 -1231.041} C_VEL
LIN {X 0,Y 594.388,Z 359.947,A -85,B 0,C 180,E1 -1233.976,E2 -1233.976} C_VEL
LIN {X 0,Y 594.391,Z 359.942,A -85,B 0,C 180,E1 -1236.296,E2 -1236.296} C_VEL
LIN {X 0,Y 594.403,Z 359.939,A -85,B 0,C 180,E1 -1239.224,E2 -1239.224} C_VEL
LIN {X 0,Y 594.378,Z 359.944,A -85,B 0,C 180,E1 -1242.095,E2 -1242.095} C_VEL
LIN {X 0,Y 594.368,Z 359.945,A -85,B 0,C 180,E1 -1244.219,E2 -1244.219} C_VEL
LIN {X 0,Y 594.367,Z 359.943,A -85,B 0,C 180,E1 -1247.017,E2 -1247.017} C_VEL
LIN {X 0,Y 594.393,Z 359.946,A -85,B 0,C 180,E1 -1249.784,E2 -1249.784} C_VEL
LIN {X 0,Y 594.391,Z 359.938,A -85,B 0,C 180,E1 -1252.526,E2 -1252.526} C_VEL
LIN {X 0,Y 594.393,Z 359.942,A -85,B 0,C 180,E1 -1255.252,E2 -1255.252} C_VEL
LIN {X 0,Y 594.394,Z 359.943,A -85,B 0,C 180,E1 -1257.967,E2 -1257.967} C_VEL
LIN {X 0,Y 594.421,Z 359.933,A -85,B 0,C 180,E1 -1260.677,E2 -1260.677} C_VEL
LIN {X 0,Y 594.381,Z 359.946,A -85,B 0,C 180,E1 -1263.389,E2 -1263.389} C_VEL
LIN {X 0,Y 594.366,Z 359.945,A -85,B 0,C 180,E1 -1266.109,E2 -1266.109} C_VEL
LIN {X 0,Y 594.395,Z 359.938,A -85,B 0,C 180,E1 -1268.842,E2 -1268.842} C_VEL
LIN {X 0,Y 594.391,Z 359.949,A -85,B 0,C 180,E1 -1271.595,E2 -1271.595} C_VEL
LIN {X 0,Y 594.387,Z 359.94,A -85,B 0,C 180,E1 -1274.377,E2 -1274.377} C_VEL
LIN {X 0,Y 594.361,Z 359.946,A -85,B 0,C 180,E1 -1275.333,E2 -1275.333} C_VEL
LIN {X 0,Y 593.688,Z 360.032,A -85,B 0,C 180,E1 -1275.899,E2 -1275.899} C_VEL
LIN {X 0,Y 590.821,Z 360.387,A -85,B 0,C 180,E1 -1276.817,E2 -1276.817} C_VEL
LIN {X 0,Y 588.41,Z 360.692,A -85,B 0,C 180,E1 -1277.555,E2 -1277.555} C_VEL
LIN {X 0,Y 587.386,Z 360.812,A -85,B 0,C 180,E1 -1278.126,E2 -1278.126} C_VEL
LIN {X 0,Y 587.309,Z 360.82,A -85,B 0,C 180,E1 -1278.319,E2 -1278.319} C_VEL
LIN {X 0,Y 587.326,Z 360.821,A -85,B 0,C 180,E1 -1281.037,E2 -1281.037} C_VEL
LIN {X 0,Y 587.319,Z 360.826,A -85,B 0,C 180,E1 -1283.258,E2 -1283.258} C_VEL
LIN {X 0,Y 587.334,Z 360.827,A -85,B 0,C 180,E1 -1285.516,E2 -1285.516} C_VEL
LIN {X 0,Y 587.345,Z 360.82,A -85,B 0,C 180,E1 -1287.817,E2 -1287.817} C_VEL
LIN {X 0,Y 587.338,Z 360.818,A -85,B 0,C 180,E1 -1290.511,E2 -1290.511} C_VEL
LIN {X 0,Y 587.337,Z 360.823,A -85,B 0,C 180,E1 -1293.112,E2 -1293.112} C_VEL
LIN {X 0,Y 587.351,Z 360.818,A -85,B 0,C 180,E1 -1295.895,E2 -1295.895} C_VEL
LIN {X 0,Y 587.328,Z 360.819,A -85,B 0,C 180,E1 -1298.479,E2 -1298.479} C_VEL
LIN {X 0,Y 587.334,Z 360.824,A -85,B 0,C 180,E1 -1301.156,E2 -1301.156} C_VEL
LIN {X 0,Y 587.33,Z 360.819,A -85,B 0,C 180,E1 -1304.114,E2 -1304.114} C_VEL
LIN {X 0,Y 587.31,Z 360.824,A -85,B 0,C 180,E1 -1306.994,E2 -1306.994} C_VEL
LIN {X 0,Y 587.316,Z 360.823,A -85,B 0,C 180,E1 -1309.746,E2 -1309.746} C_VEL
LIN {X 0,Y 587.341,Z 360.818,A -85,B 0,C 180,E1 -1312.392,E2 -1312.392} C_VEL
LIN {X 0,Y 587.349,Z 360.82,A -85,B 0,C 180,E1 -1314.946,E2 -1314.946} C_VEL
LIN {X 0,Y 587.336,Z 360.825,A -85,B 0,C 180,E1 -1317.421,E2 -1317.421} C_VEL
LIN {X 0,Y 587.344,Z 360.817,A -85,B 0,C 180,E1 -1319.831,E2 -1319.831} C_VEL
LIN {X 0,Y 587.348,Z 360.817,A -85,B 0,C 180,E1 -1322.307,E2 -1322.307} C_VEL
LIN {X 0,Y 587.333,Z 360.82,A -85,B 0,C 180,E1 -1324.483,E2 -1324.483} C_VEL
LIN {X 0,Y 587.316,Z 360.831,A -85,B 0,C 180,E1 -1327.131,E2 -1327.131} C_VEL
LIN {X 0,Y 587.327,Z 360.822,A -85,B 0,C 180,E1 -1329.695,E2 -1329.695} C_VEL
LIN {X 0,Y 587.355,Z 360.818,A -85,B 0,C 180,E1 -1332.594,E2 -1332.594} C_VEL
LIN {X 0,Y 587.362,Z 360.817,A -85,B 0,C 180,E1 -1335.739,E2 -1335.739} C_VEL
LIN {X 0,Y 587.345,Z 360.824,A -85,B 0,C 180,E1 -1338.866,E2 -1338.866} C_VEL
LIN {X 0,Y 587.363,Z 360.816,A -85,B 0,C 180,E1 -1341.745,E2 -1341.745} C_VEL
LIN {X 0,Y 587.362,Z 360.818,A -85,B 0,C 180,E1 -1344.507,E2 -1344.507} C_VEL
LIN {X 0,Y 587.368,Z 360.821,A -85,B 0,C 180,E1 -1347.257,E2 -1347.257} C_VEL
LIN {X 0,Y 587.382,Z 360.813,A -85,B 0,C 180,E1 -1350,E2 -1350} C_VEL
LIN {X 0,Y 587.368,Z 360.821,A -85,B 0,C 180,E1 -1352.743,E2 -1352.743} C_VEL
LIN {X 0,Y 587.362,Z 360.818,A -85,B 0,C 180,E1 -1355.493,E2 -1355.493} C_VEL
LIN {X 0,Y 587.367,Z 360.816,A -85,B 0,C 180,E1 -1358.255,E2 -1358.255} C_VEL
LIN {X 0,Y 587.344,Z 360.824,A -85,B 0,C 180,E1 -1361.133,E2 -1361.133} C_VEL
LIN {X 0,Y 587.361,Z 360.817,A -85,B 0,C 180,E1 -1364.261,E2 -1364.261} C_VEL
LIN {X 0,Y 587.354,Z 360.818,A -85,B 0,C 180,E1 -1367.405,E2 -1367.405} C_VEL
LIN {X 0,Y 587.327,Z 360.822,A -85,B 0,C 180,E1 -1370.304,E2 -1370.304} C_VEL
LIN {X 0,Y 587.319,Z 360.824,A -85,B 0,C 180,E1 -1373.258,E2 -1373.258} C_VEL
LIN {X 0,Y 587.333,Z 360.82,A -85,B 0,C 180,E1 -1375.516,E2 -1375.516} C_VEL
LIN {X 0,Y 587.344,Z 360.817,A -85,B 0,C 180,E1 -1377.817,E2 -1377.817} C_VEL
LIN {X 0,Y 587.346,Z 360.821,A -85,B 0,C 180,E1 -1380.512,E2 -1380.512} C_VEL
LIN {X 0,Y 587.33,Z 360.819,A -85,B 0,C 180,E1 -1383.396,E2 -1383.396} C_VEL
LIN {X 0,Y 587.352,Z 360.815,A -85,B 0,C 180,E1 -1385.895,E2 -1385.895} C_VEL
LIN {X 0,Y 587.328,Z 360.825,A -85,B 0,C 180,E1 -1388.479,E2 -1388.479} C_VEL
LIN {X 0,Y 587.331,Z 360.818,A -85,B 0,C 180,E1 -1391.156,E2 -1391.156} C_VEL
LIN {X 0,Y 587.327,Z 360.819,A -85,B 0,C 180,E1 -1394.114,E2 -1394.114} C_VEL
LIN {X 0,Y 587.33,Z 360.823,A -85,B 0,C 180,E1 -1396.996,E2 -1396.996} C_VEL
LIN {X 0,Y 587.316,Z 360.821,A -85,B 0,C 180,E1 -1399.981,E2 -1399.981} C_VEL
LIN {X 0,Y 587.34,Z 360.824,A -85,B 0,C 180,E1 -1402.393,E2 -1402.393} C_VEL
LIN {X 0,Y 587.341,Z 360.82,A -85,B 0,C 180,E1 -1404.946,E2 -1404.946} C_VEL
LIN {X 0,Y 587.337,Z 360.818,A -85,B 0,C 180,E1 -1407.421,E2 -1407.421} C_VEL
LIN {X 0,Y 587.34,Z 360.818,A -85,B 0,C 180,E1 -1409.831,E2 -1409.831} C_VEL
LIN {X 0,Y 587.344,Z 360.822,A -85,B 0,C 180,E1 -1412.307,E2 -1412.307} C_VEL
LIN {X 0,Y 587.333,Z 360.827,A -85,B 0,C 180,E1 -1414.484,E2 -1414.484} C_VEL
LIN {X 0,Y 587.336,Z 360.818,A -85,B 0,C 180,E1 -1417.487,E2 -1417.487} C_VEL
LIN {X 0,Y 587.327,Z 360.818,A -85,B 0,C 180,E1 -1419.696,E2 -1419.696} C_VEL
LIN {X 0,Y 587.353,Z 360.824,A -85,B 0,C 180,E1 -1422.595,E2 -1422.595} C_VEL
LIN {X 0,Y 587.358,Z 360.816,A -85,B 0,C 180,E1 -1425.739,E2 -1425.739} C_VEL
LIN {X 0,Y 587.337,Z 360.825,A -85,B 0,C 180,E1 -1428.263,E2 -1428.263} C_VEL
LIN {X 0,Y 587.339,Z 360.817,A -85,B 0,C 180,E1 -1431.051,E2 -1431.051} C_VEL
LIN {X 0,Y 587.369,Z 360.814,A -85,B 0,C 180,E1 -1433.264,E2 -1433.264} C_VEL
LIN {X 0,Y 587.316,Z 360.823,A -85,B 0,C 180,E1 -1435.883,E2 -1435.883} C_VEL
LIN {X 0,Y 587.364,Z 360.817,A -85,B 0,C 180,E1 -1437.943,E2 -1437.943} C_VEL
LIN {X 0,Y 587.39,Z 360.815,A -85,B 0,C 180,E1 -1440.686,E2 -1440.686} C_VEL
LIN {X 0,Y 587.331,Z 360.818,A -85,B 0,C 180,E1 -1443.43,E2 -1443.43} C_VEL
LIN {X 0,Y 587.355,Z 360.816,A -85,B 0,C 180,E1 -1445.493,E2 -1445.493} C_VEL
LIN {X 0,Y 587.366,Z 360.823,A -85,B 0,C 180,E1 -1448.256,E2 -1448.256} C_VEL
LIN {X 0,Y 587.342,Z 360.816,A -85,B 0,C 180,E1 -1451.134,E2 -1451.134} C_VEL
LIN {X 0,Y 587.355,Z 360.819,A -85,B 0,C 180,E1 -1453.846,E2 -1453.846} C_VEL
LIN {X 0,Y 587.359,Z 360.815,A -85,B 0,C 180,E1 -1456.82,E2 -1456.82} C_VEL
LIN {X 0,Y 587.341,Z 360.816,A -85,B 0,C 180,E1 -1459.575,E2 -1459.575} C_VEL
LIN {X 0,Y 587.323,Z 360.823,A -85,B 0,C 180,E1 -1461.775,E2 -1461.775} C_VEL
LIN {X 0,Y 587.348,Z 360.817,A -85,B 0,C 180,E1 -1464.759,E2 -1464.759} C_VEL
LIN {X 0,Y 587.326,Z 360.817,A -85,B 0,C 180,E1 -1467.047,E2 -1467.047} C_VEL
LIN {X 0,Y 587.348,Z 360.817,A -85,B 0,C 180,E1 -1469.38,E2 -1469.38} C_VEL
LIN {X 0,Y 587.354,Z 360.821,A -85,B 0,C 180,E1 -1471.839,E2 -1471.839} C_VEL
LIN {X 0,Y 587.351,Z 360.821,A -85,B 0,C 180,E1 -1474.35,E2 -1474.35} C_VEL
LIN {X 0,Y 587.35,Z 360.817,A -85,B 0,C 180,E1 -1476.747,E2 -1476.747} C_VEL
LIN {X 0,Y 587.344,Z 360.817,A -85,B 0,C 180,E1 -1479.36,E2 -1479.36} C_VEL
LIN {X 0,Y 587.332,Z 360.828,A -85,B 0,C 180,E1 -1482.108,E2 -1482.108} C_VEL
LIN {X 0,Y 587.314,Z 360.821,A -85,B 0,C 180,E1 -1484.912,E2 -1484.912} C_VEL
LIN {X 0,Y 587.352,Z 360.825,A -85,B 0,C 180,E1 -1487.928,E2 -1487.928} C_VEL
LIN {X 0,Y 587.334,Z 360.818,A -85,B 0,C 180,E1 -1491.059,E2 -1491.059} C_VEL
LIN {X 0,Y 587.354,Z 360.817,A -85,B 0,C 180,E1 -1493.292,E2 -1493.292} C_VEL
LIN {X 0,Y 587.369,Z 360.821,A -85,B 0,C 180,E1 -1495.781,E2 -1495.781} C_VEL
LIN {X 0,Y 587.347,Z 360.823,A -85,B 0,C 180,E1 -1498.232,E2 -1498.232} C_VEL
LIN {X 0,Y 587.352,Z 360.817,A -85,B 0,C 180,E1 -1500.867,E2 -1500.867} C_VEL
LIN {X 0,Y 587.361,Z 360.824,A -85,B 0,C 180,E1 -1503.819,E2 -1503.819} C_VEL
LIN {X 0,Y 587.387,Z 361.039,A -85,B 0,C 180,E1 -1505.413,E2 -1505.413} C_VEL
LIN {X 0,Y 587.726,Z 366.256,A -85,B 0,C 180,E1 -1506.385,E2 -1506.385} C_VEL
LIN {X 0,Y 587.597,Z 381.778,A -85,B 0,C 180,E1 -1509.156,E2 -1509.156} C_VEL
LIN {X 0,Y 587.499,Z 398.334,A -85,B 0,C 180,E1 -1512.06,E2 -1512.06} C_VEL
LIN {X 0,Y 587.402,Z 414.891,A -85,B 0,C 180,E1 -1514.917,E2 -1514.917} C_VEL
LIN {X 0,Y 587.388,Z 424.237,A -85,B 0,C 180,E1 -1516.486,E2 -1516.486} C_VEL
LIN {X 0,Y 587.759,Z 426.75,A -85,B 0,C 180,E1 -1516.561,E2 -1516.561} C_VEL
LIN {X 0,Y 587.724,Z 530.805,A -85,B 0,C 180,E1 -1517.855,E2 -1517.855} C_VEL
LIN {X 0,Y 587.695,Z 543.497,A -85,B 0,C 180,E1 -1518.139,E2 -1518.139} C_VEL
LIN {X 0,Y 587.611,Z 556.795,A -85,B 0,C 180,E1 -1518.591,E2 -1518.591} C_VEL
LIN {X 0,Y 587.555,Z 568.587,A -85,B 0,C 180,E1 -1519.141,E2 -1519.141} C_VEL
LIN {X 0,Y 587.439,Z 578.878,A -85,B 0,C 180,E1 -1519.749,E2 -1519.749} C_VEL
LIN {X 0,Y 587.376,Z 589.532,A -85,B 0,C 180,E1 -1520.531,E2 -1520.531} C_VEL
LIN {X 0,Y 587.309,Z 599.113,A -85,B 0,C 180,E1 -1521.398,E2 -1521.398} C_VEL
LIN {X 0,Y 587.271,Z 608.333,A -85,B 0,C 180,E1 -1522.436,E2 -1522.436} C_VEL
LIN {X 0,Y 587.213,Z 615.296,A -85,B 0,C 180,E1 -1523.404,E2 -1523.404} C_VEL
LIN {X 0,Y 587.211,Z 621.663,A -85,B 0,C 180,E1 -1524.506,E2 -1524.506} C_VEL
LIN {X 0,Y 587.188,Z 626.351,A -85,B 0,C 180,E1 -1525.538,E2 -1525.538} C_VEL
LIN {X 0,Y 587.194,Z 629.944,A -85,B 0,C 180,E1 -1526.569,E2 -1526.569} C_VEL
LIN {X 0,Y 587.132,Z 631.791,A -85,B 0,C 180,E1 -1527.256,E2 -1527.256} C_VEL
LIN {X 0,Y 587.139,Z 633.206,A -85,B 0,C 180,E1 -1527.942,E2 -1527.942} C_VEL
LIN {X 0,Y 587.14,Z 634.785,A -85,B 0,C 180,E1 -1529.314,E2 -1529.314} C_VEL
LIN {X 0,Y 587.137,Z 635,A -85,B 0,C 180,E1 -1530,E2 -1530} C_VEL
LIN {X 0,Y 587.147,Z 634.182,A -85,B 0,C 180,E1 -1531.372,E2 -1531.372} C_VEL
LIN {X 0,Y 587.139,Z 633.205,A -85,B 0,C 180,E1 -1532.058,E2 -1532.058} C_VEL
LIN {X 0,Y 587.132,Z 631.79,A -85,B 0,C 180,E1 -1532.745,E2 -1532.745} C_VEL
LIN {X 0,Y 587.212,Z 628.873,A -85,B 0,C 180,E1 -1533.774,E2 -1533.774} C_VEL
LIN {X 0,Y 587.147,Z 624.93,A -85,B 0,C 180,E1 -1534.806,E2 -1534.806} C_VEL
LIN {X 0,Y 587.229,Z 619.854,A -85,B 0,C 180,E1 -1535.839,E2 -1535.839} C_VEL
LIN {X 0,Y 587.245,Z 612.238,A -85,B 0,C 180,E1 -1537.046,E2 -1537.046} C_VEL
LIN {X 0,Y 587.299,Z 603.965,A -85,B 0,C 180,E1 -1538.083,E2 -1538.083} C_VEL
LIN {X 0,Y 587.343,Z 595.497,A -85,B 0,C 180,E1 -1538.949,E2 -1538.949} C_VEL
LIN {X 0,Y 587.413,Z 585.098,A -85,B 0,C 180,E1 -1539.816,E2 -1539.816} C_VEL
LIN {X 0,Y 587.515,Z 573.306,A -85,B 0,C 180,E1 -1540.598,E2 -1540.598} C_VEL
LIN {X 0,Y 587.581,Z 562.773,A -85,B 0,C 180,E1 -1541.147,E2 -1541.147} C_VEL
LIN {X 0,Y 587.629,Z 551.887,A -85,B 0,C 180,E1 -1541.593,E2 -1541.593} C_VEL
LIN {X 0,Y 587.706,Z 540.107,A -85,B 0,C 180,E1 -1541.948,E2 -1541.948} C_VEL
LIN {X 0,Y 587.759,Z 528.104,A -85,B 0,C 180,E1 -1542.188,E2 -1542.188} C_VEL
LIN {X 0,Y 587.743,Z 426.716,A -85,B 0,C 180,E1 -1543.44,E2 -1543.44} C_VEL
LIN {X 0,Y 587.389,Z 424.234,A -85,B 0,C 180,E1 -1543.514,E2 -1543.514} C_VEL
LIN {X 0,Y 587.448,Z 408.68,A -85,B 0,C 180,E1 -1546.15,E2 -1546.15} C_VEL
LIN {X 0,Y 587.52,Z 393.158,A -85,B 0,C 180,E1 -1548.843,E2 -1548.843} C_VEL
LIN {X 0,Y 587.635,Z 376.601,A -85,B 0,C 180,E1 -1551.762,E2 -1551.762} C_VEL
LIN {X 0,Y 587.752,Z 364.184,A -85,B 0,C 180,E1 -1553.988,E2 -1553.988} C_VEL
LIN {X 0,Y 587.371,Z 360.904,A -85,B 0,C 180,E1 -1554.631,E2 -1554.631} C_VEL
LIN {X 0,Y 587.332,Z 360.82,A -85,B 0,C 180,E1 -1557.046,E2 -1557.046} C_VEL
LIN {X 0,Y 587.354,Z 360.817,A -85,B 0,C 180,E1 -1559.379,E2 -1559.379} C_VEL
LIN {X 0,Y 587.347,Z 360.824,A -85,B 0,C 180,E1 -1561.835,E2 -1561.835} C_VEL
LIN {X 0,Y 587.359,Z 360.82,A -85,B 0,C 180,E1 -1564.349,E2 -1564.349} C_VEL
LIN {X 0,Y 587.355,Z 360.816,A -85,B 0,C 180,E1 -1566.746,E2 -1566.746} C_VEL
LIN {X 0,Y 587.348,Z 360.818,A -85,B 0,C 180,E1 -1569.359,E2 -1569.359} C_VEL
LIN {X 0,Y 587.336,Z 360.826,A -85,B 0,C 180,E1 -1572.107,E2 -1572.107} C_VEL
LIN {X 0,Y 587.317,Z 360.82,A -85,B 0,C 180,E1 -1575.088,E2 -1575.088} C_VEL
LIN {X 0,Y 587.354,Z 360.826,A -85,B 0,C 180,E1 -1577.927,E2 -1577.927} C_VEL
LIN {X 0,Y 587.334,Z 360.818,A -85,B 0,C 180,E1 -1581.058,E2 -1581.058} C_VEL
LIN {X 0,Y 587.354,Z 360.817,A -85,B 0,C 180,E1 -1583.291,E2 -1583.291} C_VEL
LIN {X 0,Y 587.362,Z 360.822,A -85,B 0,C 180,E1 -1585.78,E2 -1585.78} C_VEL
LIN {X 0,Y 587.353,Z 360.82,A -85,B 0,C 180,E1 -1588.231,E2 -1588.231} C_VEL
LIN {X 0,Y 587.35,Z 360.816,A -85,B 0,C 180,E1 -1590.866,E2 -1590.866} C_VEL
LIN {X 0,Y 587.36,Z 360.823,A -85,B 0,C 180,E1 -1593.818,E2 -1593.818} C_VEL
LIN {X 0,Y 587.338,Z 360.825,A -85,B 0,C 180,E1 -1595.993,E2 -1595.993} C_VEL
LIN {X 0,Y 587.325,Z 360.822,A -85,B 0,C 180,E1 -1598.225,E2 -1598.225} C_VEL
LIN {X 0,Y 587.348,Z 360.816,A -85,B 0,C 180,E1 -1601.151,E2 -1601.151} C_VEL
LIN {X 0,Y 587.352,Z 360.817,A -85,B 0,C 180,E1 -1603.311,E2 -1603.311} C_VEL
LIN {X 0,Y 587.358,Z 360.819,A -85,B 0,C 180,E1 -1606.154,E2 -1606.154} C_VEL
LIN {X 0,Y 587.341,Z 360.817,A -85,B 0,C 180,E1 -1608.962,E2 -1608.962} C_VEL
LIN {X 0,Y 587.368,Z 360.822,A -85,B 0,C 180,E1 -1611.744,E2 -1611.744} C_VEL
LIN {X 0,Y 587.356,Z 360.816,A -85,B 0,C 180,E1 -1614.507,E2 -1614.507} C_VEL
LIN {X 0,Y 587.376,Z 360.816,A -85,B 0,C 180,E1 -1617.256,E2 -1617.256} C_VEL
LIN {X 0,Y 587.381,Z 360.814,A -85,B 0,C 180,E1 -1620,E2 -1620} C_VEL
LIN {X 0,Y 587.376,Z 360.812,A -85,B 0,C 180,E1 -1622.743,E2 -1622.743} C_VEL
LIN {X 0,Y 587.355,Z 360.824,A -85,B 0,C 180,E1 -1625.493,E2 -1625.493} C_VEL
LIN {X 0,Y 587.368,Z 360.814,A -85,B 0,C 180,E1 -1628.255,E2 -1628.255} C_VEL
LIN {X 0,Y 587.344,Z 360.818,A -85,B 0,C 180,E1 -1631.133,E2 -1631.133} C_VEL
LIN {X 0,Y 587.361,Z 360.816,A -85,B 0,C 180,E1 -1634.26,E2 -1634.26} C_VEL
LIN {X 0,Y 587.349,Z 360.824,A -85,B 0,C 180,E1 -1637.406,E2 -1637.406} C_VEL
LIN {X 0,Y 587.309,Z 360.82,A -85,B 0,C 180,E1 -1638.319,E2 -1638.319} C_VEL
LIN {X 0,Y 586.665,Z 360.902,A -85,B 0,C 180,E1 -1638.891,E2 -1638.891} C_VEL
LIN {X 0,Y 583.837,Z 361.259,A -85,B 0,C 180,E1 -1639.819,E2 -1639.819} C_VEL
LIN {X 0,Y 581.426,Z 361.563,A -85,B 0,C 180,E1 -1640.566,E2 -1640.566} C_VEL
LIN {X 0,Y 580.373,Z 361.692,A -85,B 0,C 180,E1 -1641.143,E2 -1641.143} C_VEL
LIN {X 0,Y 580.279,Z 361.702,A -85,B 0,C 180,E1 -1641.338,E2 -1641.338} C_VEL
LIN {X 0,Y 580.297,Z 361.695,A -85,B 0,C 180,E1 -1644.316,E2 -1644.316} C_VEL
LIN {X 0,Y 580.303,Z 361.693,A -85,B 0,C 180,E1 -1646.622,E2 -1646.622} C_VEL
LIN {X 0,Y 580.299,Z 361.701,A -85,B 0,C 180,E1 -1649.31,E2 -1649.31} C_VEL
LIN {X 0,Y 580.3,Z 361.695,A -85,B 0,C 180,E1 -1652.2,E2 -1652.2} C_VEL
LIN {X 0,Y 580.295,Z 361.694,A -85,B 0,C 180,E1 -1654.695,E2 -1654.695} C_VEL
LIN {X 0,Y 580.297,Z 361.703,A -85,B 0,C 180,E1 -1657.268,E2 -1657.268} C_VEL
LIN {X 0,Y 580.294,Z 361.694,A -85,B 0,C 180,E1 -1660.271,E2 -1660.271} C_VEL
LIN {X 0,Y 580.279,Z 361.698,A -85,B 0,C 180,E1 -1662.706,E2 -1662.706} C_VEL
LIN {X 0,Y 580.265,Z 361.702,A -85,B 0,C 180,E1 -1665.609,E2 -1665.609} C_VEL
LIN {X 0,Y 580.294,Z 361.69,A -85,B 0,C 180,E1 -1668.233,E2 -1668.233} C_VEL
LIN {X 0,Y 580.286,Z 361.7,A -85,B 0,C 180,E1 -1670.966,E2 -1670.966} C_VEL
LIN {X 0,Y 580.293,Z 361.699,A -85,B 0,C 180,E1 -1673.598,E2 -1673.598} C_VEL
LIN {X 0,Y 580.316,Z 361.691,A -85,B 0,C 180,E1 -1676.146,E2 -1676.146} C_VEL
LIN {X 0,Y 580.286,Z 361.698,A -85,B 0,C 180,E1 -1678.615,E2 -1678.615} C_VEL
LIN {X 0,Y 580.292,Z 361.701,A -85,B 0,C 180,E1 -1681.024,E2 -1681.024} C_VEL
LIN {X 0,Y 580.289,Z 361.699,A -85,B 0,C 180,E1 -1683.666,E2 -1683.666} C_VEL
LIN {X 0,Y 580.298,Z 361.698,A -85,B 0,C 180,E1 -1685.684,E2 -1685.684} C_VEL
LIN {X 0,Y 580.27,Z 361.699,A -85,B 0,C 180,E1 -1687.947,E2 -1687.947} C_VEL
LIN {X 0,Y 580.316,Z 361.7,A -85,B 0,C 180,E1 -1690.914,E2 -1690.914} C_VEL
LIN {X 0,Y 580.276,Z 361.699,A -85,B 0,C 180,E1 -1693.825,E2 -1693.825} C_VEL
LIN {X 0,Y 580.324,Z 361.692,A -85,B 0,C 180,E1 -1695.983,E2 -1695.983} C_VEL
LIN {X 0,Y 580.301,Z 361.701,A -85,B 0,C 180,E1 -1698.827,E2 -1698.827} C_VEL
LIN {X 0,Y 580.326,Z 361.694,A -85,B 0,C 180,E1 -1701.644,E2 -1701.644} C_VEL
LIN {X 0,Y 580.329,Z 361.693,A -85,B 0,C 180,E1 -1704.44,E2 -1704.44} C_VEL
LIN {X 0,Y 580.335,Z 361.698,A -85,B 0,C 180,E1 -1707.223,E2 -1707.223} C_VEL
LIN {X 0,Y 580.351,Z 361.689,A -85,B 0,C 180,E1 -1710,E2 -1710} C_VEL
LIN {X 0,Y 580.335,Z 361.698,A -85,B 0,C 180,E1 -1712.776,E2 -1712.776} C_VEL
LIN {X 0,Y 580.329,Z 361.693,A -85,B 0,C 180,E1 -1715.559,E2 -1715.559} C_VEL
LIN {X 0,Y 580.33,Z 361.693,A -85,B 0,C 180,E1 -1718.356,E2 -1718.356} C_VEL
LIN {X 0,Y 580.296,Z 361.701,A -85,B 0,C 180,E1 -1721.191,E2 -1721.191} C_VEL
LIN {X 0,Y 580.323,Z 361.692,A -85,B 0,C 180,E1 -1724.017,E2 -1724.017} C_VEL
LIN {X 0,Y 580.308,Z 361.704,A -85,B 0,C 180,E1 -1726.914,E2 -1726.914} C_VEL
LIN {X 0,Y 580.301,Z 361.695,A -85,B 0,C 180,E1 -1729.822,E2 -1729.822} C_VEL
LIN {X 0,Y 580.291,Z 361.706,A -85,B 0,C 180,E1 -1732.802,E2 -1732.802} C_VEL
LIN {X 0,Y 580.303,Z 361.7,A -85,B 0,C 180,E1 -1735.079,E2 -1735.079} C_VEL
LIN {X 0,Y 580.315,Z 361.693,A -85,B 0,C 180,E1 -1737.863,E2 -1737.863} C_VEL
LIN {X 0,Y 580.295,Z 361.703,A -85,B 0,C 180,E1 -1740.697,E2 -1740.697} C_VEL
LIN {X 0,Y 580.299,Z 361.695,A -85,B 0,C 180,E1 -1743.316,E2 -1743.316} C_VEL
LIN {X 0,Y 580.322,Z 361.69,A -85,B 0,C 180,E1 -1745.768,E2 -1745.768} C_VEL
LIN {X 0,Y 580.284,Z 361.699,A -85,B 0,C 180,E1 -1748.146,E2 -1748.146} C_VEL
LIN {X 0,Y 580.294,Z 361.698,A -85,B 0,C 180,E1 -1750.843,E2 -1750.843} C_VEL
LIN {X 0,Y 580.28,Z 361.695,A -85,B 0,C 180,E1 -1753.657,E2 -1753.657} C_VEL
LIN {X 0,Y 580.285,Z 361.706,A -85,B 0,C 180,E1 -1756.607,E2 -1756.607} C_VEL
LIN {X 0,Y 580.295,Z 361.696,A -85,B 0,C 180,E1 -1759.157,E2 -1759.157} C_VEL
LIN {X 0,Y 580.284,Z 361.697,A -85,B 0,C 180,E1 -1761.927,E2 -1761.927} C_VEL
LIN {X 0,Y 580.299,Z 361.702,A -85,B 0,C 180,E1 -1764.457,E2 -1764.457} C_VEL
LIN {X 0,Y 580.286,Z 361.7,A -85,B 0,C 180,E1 -1766.975,E2 -1766.975} C_VEL
LIN {X 0,Y 580.303,Z 361.694,A -85,B 0,C 180,E1 -1769.426,E2 -1769.426} C_VEL
LIN {X 0,Y 580.313,Z 361.695,A -85,B 0,C 180,E1 -1772.137,E2 -1772.137} C_VEL
LIN {X 0,Y 580.302,Z 361.698,A -85,B 0,C 180,E1 -1774.921,E2 -1774.921} C_VEL
LIN {X 0,Y 580.27,Z 361.7,A -85,B 0,C 180,E1 -1777.948,E2 -1777.948} C_VEL
LIN {X 0,Y 580.311,Z 361.694,A -85,B 0,C 180,E1 -1780.914,E2 -1780.914} C_VEL
LIN {X 0,Y 580.278,Z 361.698,A -85,B 0,C 180,E1 -1783.826,E2 -1783.826} C_VEL
LIN {X 0,Y 580.32,Z 361.695,A -85,B 0,C 180,E1 -1785.983,E2 -1785.983} C_VEL
LIN {X 0,Y 580.297,Z 361.696,A -85,B 0,C 180,E1 -1788.827,E2 -1788.827} C_VEL
LIN {X 0,Y 580.329,Z 361.689,A -85,B 0,C 180,E1 -1791.644,E2 -1791.644} C_VEL
LIN {X 0,Y 580.32,Z 361.702,A -85,B 0,C 180,E1 -1794.441,E2 -1794.441} C_VEL
LIN {X 0,Y 580.34,Z 361.688,A -85,B 0,C 180,E1 -1797.224,E2 -1797.224} C_VEL
LIN {X 0,Y 580.347,Z 361.689,A -85,B 0,C 180,E1 -1800,E2 -1800} C_VEL
LIN {X 0,Y 580.34,Z 361.692,A -85,B 0,C 180,E1 -1802.777,E2 -1802.777} C_VEL
LIN {X 0,Y 580.321,Z 361.692,A -85,B 0,C 180,E1 -1805.56,E2 -1805.56} C_VEL
LIN {X 0,Y 580.33,Z 361.696,A -85,B 0,C 180,E1 -1808.356,E2 -1808.356} C_VEL
LIN {X 0,Y 580.294,Z 361.694,A -85,B 0,C 180,E1 -1811.192,E2 -1811.192} C_VEL
LIN {X 0,Y 580.321,Z 361.698,A -85,B 0,C 180,E1 -1814.017,E2 -1814.017} C_VEL
LIN {X 0,Y 580.309,Z 361.692,A -85,B 0,C 180,E1 -1816.915,E2 -1816.915} C_VEL
LIN {X 0,Y 580.303,Z 361.695,A -85,B 0,C 180,E1 -1819.823,E2 -1819.823} C_VEL
LIN {X 0,Y 580.273,Z 361.705,A -85,B 0,C 180,E1 -1822.053,E2 -1822.053} C_VEL
LIN {X 0,Y 580.304,Z 361.693,A -85,B 0,C 180,E1 -1825.08,E2 -1825.08} C_VEL
LIN {X 0,Y 580.316,Z 361.695,A -85,B 0,C 180,E1 -1827.864,E2 -1827.864} C_VEL
LIN {X 0,Y 580.296,Z 361.697,A -85,B 0,C 180,E1 -1830.698,E2 -1830.698} C_VEL
LIN {X 0,Y 580.303,Z 361.693,A -85,B 0,C 180,E1 -1833.318,E2 -1833.318} C_VEL
LIN {X 0,Y 580.322,Z 361.696,A -85,B 0,C 180,E1 -1835.768,E2 -1835.768} C_VEL
LIN {X 0,Y 580.288,Z 361.705,A -85,B 0,C 180,E1 -1838.147,E2 -1838.147} C_VEL
LIN {X 0,Y 580.299,Z 361.695,A -85,B 0,C 180,E1 -1840.844,E2 -1840.844} C_VEL
LIN {X 0,Y 580.287,Z 361.7,A -85,B 0,C 180,E1 -1843.658,E2 -1843.658} C_VEL
LIN {X 0,Y 580.275,Z 361.699,A -85,B 0,C 180,E1 -1846.61,E2 -1846.61} C_VEL
LIN {X 0,Y 580.299,Z 361.692,A -85,B 0,C 180,E1 -1849.158,E2 -1849.158} C_VEL
LIN {X 0,Y 580.291,Z 361.705,A -85,B 0,C 180,E1 -1851.927,E2 -1851.927} C_VEL
LIN {X 0,Y 580.308,Z 361.696,A -85,B 0,C 180,E1 -1854.457,E2 -1854.457} C_VEL
LIN {X 0,Y 580.291,Z 361.695,A -85,B 0,C 180,E1 -1856.976,E2 -1856.976} C_VEL
LIN {X 0,Y 580.308,Z 361.697,A -85,B 0,C 180,E1 -1859.426,E2 -1859.426} C_VEL
LIN {X 0,Y 580.321,Z 361.7,A -85,B 0,C 180,E1 -1862.138,E2 -1862.138} C_VEL
LIN {X 0,Y 580.334,Z 361.834,A -85,B 0,C 180,E1 -1865.241,E2 -1865.241} C_VEL
LIN {X 0,Y 580.805,Z 366.256,A -85,B 0,C 180,E1 -1866.087,E2 -1866.087} C_VEL
LIN {X 0,Y 580.646,Z 380.959,A -85,B 0,C 180,E1 -1868.748,E2 -1868.748} C_VEL
LIN {X 0,Y 580.517,Z 395.23,A -85,B 0,C 180,E1 -1871.288,E2 -1871.288} C_VEL
LIN {X 0,Y 580.401,Z 410.752,A -85,B 0,C 180,E1 -1874.01,E2 -1874.01} C_VEL
LIN {X 0,Y 580.359,Z 424.241,A -85,B 0,C 180,E1 -1876.319,E2 -1876.319} C_VEL
LIN {X 0,Y 580.68,Z 426.75,A -85,B 0,C 180,E1 -1876.394,E2 -1876.394} C_VEL
LIN {X 0,Y 580.967,Z 430.327,A -85,B 0,C 180,E1 -1876.445,E2 -1876.445} C_VEL
LIN {X 0,Y 580.806,Z 530.75,A -85,B 0,C 180,E1 -1877.708,E2 -1877.708} C_VEL
LIN {X 0,Y 580.769,Z 543.502,A -85,B 0,C 180,E1 -1877.996,E2 -1877.996} C_VEL
LIN {X 0,Y 580.635,Z 557.482,A -85,B 0,C 180,E1 -1878.48,E2 -1878.48} C_VEL
LIN {X 0,Y 580.562,Z 568.572,A -85,B 0,C 180,E1 -1879.009,E2 -1879.009} C_VEL
LIN {X 0,Y 580.447,Z 578.864,A -85,B 0,C 180,E1 -1879.624,E2 -1879.624} C_VEL
LIN {X 0,Y 580.369,Z 588.442,A -85,B 0,C 180,E1 -1880.328,E2 -1880.328} C_VEL
LIN {X 0,Y 580.304,Z 597.333,A -85,B 0,C 180,E1 -1881.118,E2 -1881.118} C_VEL
LIN {X 0,Y 580.221,Z 606.964,A -85,B 0,C 180,E1 -1882.168,E2 -1882.168} C_VEL
LIN {X 0,Y 580.15,Z 614.669,A -85,B 0,C 180,E1 -1883.226,E2 -1883.226} C_VEL
LIN {X 0,Y 580.161,Z 619.853,A -85,B 0,C 180,E1 -1884.09,E2 -1884.09} C_VEL
LIN {X 0,Y 580.053,Z 624.925,A -85,B 0,C 180,E1 -1885.135,E2 -1885.135} C_VEL
LIN {X 0,Y 580.109,Z 628.867,A -85,B 0,C 180,E1 -1886.18,E2 -1886.18} C_VEL
LIN {X 0,Y 580.043,Z 631.783,A -85,B 0,C 180,E1 -1887.222,E2 -1887.222} C_VEL
LIN {X 0,Y 580.039,Z 633.207,A -85,B 0,C 180,E1 -1887.917,E2 -1887.917} C_VEL
LIN {X 0,Y 580.04,Z 634.78,A -85,B 0,C 180,E1 -1889.306,E2 -1889.306} C_VEL
LIN {X 0,Y 580.037,Z 635,A -85,B 0,C 180,E1 -1890,E2 -1890} C_VEL
LIN {X 0,Y 580.047,Z 634.182,A -85,B 0,C 180,E1 -1891.389,E2 -1891.389} C_VEL
LIN {X 0,Y 580.038,Z 633.207,A -85,B 0,C 180,E1 -1892.083,E2 -1892.083} C_VEL
LIN {X 0,Y 580.043,Z 631.782,A -85,B 0,C 180,E1 -1892.778,E2 -1892.778} C_VEL
LIN {X 0,Y 580.109,Z 628.866,A -85,B 0,C 180,E1 -1893.821,E2 -1893.821} C_VEL
LIN {X 0,Y 580.053,Z 624.924,A -85,B 0,C 180,E1 -1894.865,E2 -1894.865} C_VEL
LIN {X 0,Y 580.161,Z 619.851,A -85,B 0,C 180,E1 -1895.91,E2 -1895.91} C_VEL
LIN {X 0,Y 580.184,Z 612.24,A -85,B 0,C 180,E1 -1897.132,E2 -1897.132} C_VEL
LIN {X 0,Y 580.25,Z 603.954,A -85,B 0,C 180,E1 -1898.182,E2 -1898.182} C_VEL
LIN {X 0,Y 580.308,Z 595.484,A -85,B 0,C 180,E1 -1899.058,E2 -1899.058} C_VEL
LIN {X 0,Y 580.388,Z 586.246,A -85,B 0,C 180,E1 -1899.848,E2 -1899.848} C_VEL
LIN {X 0,Y 580.509,Z 574.773,A -85,B 0,C 180,E1 -1900.639,E2 -1900.639} C_VEL
LIN {X 0,Y 580.593,Z 563.324,A -85,B 0,C 180,E1 -1901.258,E2 -1901.258} C_VEL
LIN {X 0,Y 580.681,Z 551.661,A -85,B 0,C 180,E1 -1901.741,E2 -1901.741} C_VEL
LIN {X 0,Y 580.775,Z 540.073,A -85,B 0,C 180,E1 -1902.093,E2 -1902.093} C_VEL
LIN {X 0,Y 580.835,Z 528.082,A -85,B 0,C 180,E1 -1902.336,E2 -1902.336} C_VEL
LIN {X 0,Y 580.839,Z 427.498,A -85,B 0,C 180,E1 -1903.593,E2 -1903.593} C_VEL
LIN {X 0,Y 580.385,Z 424.548,A -85,B 0,C 180,E1 -1903.658,E2 -1903.658} C_VEL
LIN {X 0,Y 580.327,Z 422.132,A -85,B 0,C 180,E1 -1904.017,E2 -1904.017} C_VEL
LIN {X 0,Y 580.421,Z 405.575,A -85,B 0,C 180,E1 -1906.894,E2 -1906.894} C_VEL
LIN {X 0,Y 580.566,Z 390.982,A -85,B 0,C 180,E1 -1909.464,E2 -1909.464} C_VEL
LIN {X 0,Y 580.717,Z 374.532,A -85,B 0,C 180,E1 -1912.409,E2 -1912.409} C_VEL
LIN {X 0,Y 580.759,Z 364.174,A -85,B 0,C 180,E1 -1914.296,E2 -1914.296} C_VEL
LIN {X 0,Y 580.331,Z 361.75,A -85,B 0,C 180,E1 -1914.813,E2 -1914.813} C_VEL
LIN {X 0,Y 580.323,Z 361.7,A -85,B 0,C 180,E1 -1917.863,E2 -1917.863} C_VEL
LIN {X 0,Y 580.294,Z 361.698,A -85,B 0,C 180,E1 -1920.695,E2 -1920.695} C_VEL
LIN {X 0,Y 580.306,Z 361.694,A -85,B 0,C 180,E1 -1923.316,E2 -1923.316} C_VEL
LIN {X 0,Y 580.328,Z 361.697,A -85,B 0,C 180,E1 -1925.767,E2 -1925.767} C_VEL
LIN {X 0,Y 580.291,Z 361.704,A -85,B 0,C 180,E1 -1928.146,E2 -1928.146} C_VEL
LIN {X 0,Y 580.301,Z 361.692,A -85,B 0,C 180,E1 -1930.843,E2 -1930.843} C_VEL
LIN {X 0,Y 580.28,Z 361.702,A -85,B 0,C 180,E1 -1933.657,E2 -1933.657} C_VEL
LIN {X 0,Y 580.287,Z 361.697,A -85,B 0,C 180,E1 -1936.608,E2 -1936.608} C_VEL
LIN {X 0,Y 580.301,Z 361.695,A -85,B 0,C 180,E1 -1939.156,E2 -1939.156} C_VEL
LIN {X 0,Y 580.291,Z 361.706,A -85,B 0,C 180,E1 -1941.926,E2 -1941.926} C_VEL
LIN {X 0,Y 580.285,Z 361.697,A -85,B 0,C 180,E1 -1944.455,E2 -1944.455} C_VEL
LIN {X 0,Y 580.292,Z 361.694,A -85,B 0,C 180,E1 -1946.975,E2 -1946.975} C_VEL
LIN {X 0,Y 580.309,Z 361.697,A -85,B 0,C 180,E1 -1949.426,E2 -1949.426} C_VEL
LIN {X 0,Y 580.319,Z 361.695,A -85,B 0,C 180,E1 -1952.137,E2 -1952.137} C_VEL
LIN {X 0,Y 580.321,Z 361.693,A -85,B 0,C 180,E1 -1955.269,E2 -1955.269} C_VEL
LIN {X 0,Y 580.275,Z 361.705,A -85,B 0,C 180,E1 -1957.947,E2 -1957.947} C_VEL
LIN {X 0,Y 580.317,Z 361.69,A -85,B 0,C 180,E1 -1960.914,E2 -1960.914} C_VEL
LIN {X 0,Y 580.28,Z 361.706,A -85,B 0,C 180,E1 -1963.825,E2 -1963.825} C_VEL
LIN {X 0,Y 580.324,Z 361.697,A -85,B 0,C 180,E1 -1965.983,E2 -1965.983} C_VEL
LIN {X 0,Y 580.302,Z 361.693,A -85,B 0,C 180,E1 -1968.826,E2 -1968.826} C_VEL
LIN {X 0,Y 580.332,Z 361.696,A -85,B 0,C 180,E1 -1971.644,E2 -1971.644} C_VEL
LIN {X 0,Y 580.322,Z 361.692,A -85,B 0,C 180,E1 -1974.44,E2 -1974.44} C_VEL
LIN {X 0,Y 580.341,Z 361.692,A -85,B 0,C 180,E1 -1977.223,E2 -1977.223} C_VEL
LIN {X 0,Y 580.35,Z 361.689,A -85,B 0,C 180,E1 -1980,E2 -1980} C_VEL
LIN {X 0,Y 580.341,Z 361.688,A -85,B 0,C 180,E1 -1982.776,E2 -1982.776} C_VEL
LIN {X 0,Y 580.321,Z 361.701,A -85,B 0,C 180,E1 -1985.559,E2 -1985.559} C_VEL
LIN {X 0,Y 580.331,Z 361.689,A -85,B 0,C 180,E1 -1988.356,E2 -1988.356} C_VEL
LIN {X 0,Y 580.296,Z 361.696,A -85,B 0,C 180,E1 -1991.191,E2 -1991.191} C_VEL
LIN {X 0,Y 580.323,Z 361.695,A -85,B 0,C 180,E1 -1994.017,E2 -1994.017} C_VEL
LIN {X 0,Y 580.309,Z 361.694,A -85,B 0,C 180,E1 -1996.914,E2 -1996.914} C_VEL
LIN {X 0,Y 580.303,Z 361.697,A -85,B 0,C 180,E1 -1999.822,E2 -1999.822} C_VEL
LIN {X 0,Y 580.279,Z 361.702,A -85,B 0,C 180,E1 -2001.338,E2 -2001.338} C_VEL
LIN {X 0,Y 579.584,Z 361.787,A -85,B 0,C 180,E1 -2001.917,E2 -2001.917} C_VEL
LIN {X 0,Y 576.708,Z 362.143,A -85,B 0,C 180,E1 -2002.857,E2 -2002.857} C_VEL
LIN {X 0,Y 574.313,Z 362.448,A -85,B 0,C 180,E1 -2003.613,E2 -2003.613} C_VEL
LIN {X 0,Y 573.313,Z 362.566,A -85,B 0,C 180,E1 -2004.197,E2 -2004.197} C_VEL
LIN {X 0,Y 573.247,Z 362.573,A -85,B 0,C 180,E1 -2004.395,E2 -2004.395} C_VEL
LIN {X 0,Y 573.261,Z 362.572,A -85,B 0,C 180,E1 -2006.975,E2 -2006.975} C_VEL
LIN {X 0,Y 573.245,Z 362.583,A -85,B 0,C 180,E1 -2009.488,E2 -2009.488} C_VEL
LIN {X 0,Y 573.253,Z 362.572,A -85,B 0,C 180,E1 -2012.229,E2 -2012.229} C_VEL
LIN {X 0,Y 573.245,Z 362.572,A -85,B 0,C 180,E1 -2014.773,E2 -2014.773} C_VEL
LIN {X 0,Y 573.25,Z 362.579,A -85,B 0,C 180,E1 -2017.166,E2 -2017.166} C_VEL
LIN {X 0,Y 573.243,Z 362.578,A -85,B 0,C 180,E1 -2019.607,E2 -2019.607} C_VEL
LIN {X 0,Y 573.24,Z 362.575,A -85,B 0,C 180,E1 -2022.642,E2 -2022.642} C_VEL
LIN {X 0,Y 573.231,Z 362.577,A -85,B 0,C 180,E1 -2025.666,E2 -2025.666} C_VEL
LIN {X 0,Y 573.235,Z 362.569,A -85,B 0,C 180,E1 -2028.544,E2 -2028.544} C_VEL
LIN {X 0,Y 573.246,Z 362.583,A -85,B 0,C 180,E1 -2031.299,E2 -2031.299} C_VEL
LIN {X 0,Y 573.261,Z 362.57,A -85,B 0,C 180,E1 -2034.011,E2 -2034.011} C_VEL
LIN {X 0,Y 573.281,Z 362.568,A -85,B 0,C 180,E1 -2036.519,E2 -2036.519} C_VEL
LIN {X 0,Y 573.241,Z 362.583,A -85,B 0,C 180,E1 -2039.115,E2 -2039.115} C_VEL
LIN {X 0,Y 573.261,Z 362.572,A -85,B 0,C 180,E1 -2041.968,E2 -2041.968} C_VEL
LIN {X 0,Y 573.252,Z 362.575,A -85,B 0,C 180,E1 -2044.59,E2 -2044.59} C_VEL
LIN {X 0,Y 573.234,Z 362.578,A -85,B 0,C 180,E1 -2047.662,E2 -2047.662} C_VEL
LIN {X 0,Y 573.275,Z 362.574,A -85,B 0,C 180,E1 -2050.728,E2 -2050.728} C_VEL
LIN {X 0,Y 573.248,Z 362.576,A -85,B 0,C 180,E1 -2053.622,E2 -2053.622} C_VEL
LIN {X 0,Y 573.271,Z 362.572,A -85,B 0,C 180,E1 -2055.807,E2 -2055.807} C_VEL
LIN {X 0,Y 573.259,Z 362.577,A -85,B 0,C 180,E1 -2058.745,E2 -2058.745} C_VEL
LIN {X 0,Y 573.282,Z 362.573,A -85,B 0,C 180,E1 -2061.54,E2 -2061.54} C_VEL
LIN {X 0,Y 573.297,Z 362.569,A -85,B 0,C 180,E1 -2064.372,E2 -2064.372} C_VEL
LIN {X 0,Y 573.312,Z 362.566,A -85,B 0,C 180,E1 -2067.892,E2 -2067.892} C_VEL
LIN {X 0,Y 573.329,Z 362.569,A -85,B 0,C 180,E1 -2070.702,E2 -2070.702} C_VEL
LIN {X 0,Y 573.301,Z 362.575,A -85,B 0,C 180,E1 -2072.81,E2 -2072.81} C_VEL
LIN {X 0,Y 573.297,Z 362.569,A -85,B 0,C 180,E1 -2075.628,E2 -2075.628} C_VEL
LIN {X 0,Y 573.286,Z 362.572,A -85,B 0,C 180,E1 -2078.459,E2 -2078.459} C_VEL
LIN {X 0,Y 573.268,Z 362.575,A -85,B 0,C 180,E1 -2081.312,E2 -2081.312} C_VEL
LIN {X 0,Y 573.278,Z 362.573,A -85,B 0,C 180,E1 -2084.424,E2 -2084.424} C_VEL
LIN {X 0,Y 573.255,Z 362.579,A -85,B 0,C 180,E1 -2087.111,E2 -2087.111} C_VEL
LIN {X 0,Y 573.249,Z 362.574,A -85,B 0,C 180,E1 -2090.076,E2 -2090.076} C_VEL
LIN {X 0,Y 573.229,Z 362.582,A -85,B 0,C 180,E1 -2093.099,E2 -2093.099} C_VEL
LIN {X 0,Y 573.251,Z 362.575,A -85,B 0,C 180,E1 -2095.41,E2 -2095.41} C_VEL
LIN {X 0,Y 573.259,Z 362.572,A -85,B 0,C 180,E1 -2098.031,E2 -2098.031} C_VEL
LIN {X 0,Y 573.239,Z 362.583,A -85,B 0,C 180,E1 -2100.885,E2 -2100.885} C_VEL
LIN {X 0,Y 573.256,Z 362.571,A -85,B 0,C 180,E1 -2103.524,E2 -2103.524} C_VEL
LIN {X 0,Y 573.256,Z 362.571,A -85,B 0,C 180,E1 -2106.048,E2 -2106.048} C_VEL
LIN {X 0,Y 573.244,Z 362.584,A -85,B 0,C 180,E1 -2108.701,E2 -2108.701} C_VEL
LIN {X 0,Y 573.237,Z 362.569,A -85,B 0,C 180,E1 -2111.594,E2 -2111.594} C_VEL
LIN {X 0,Y 573.232,Z 362.577,A -85,B 0,C 180,E1 -2114.333,E2 -2114.333} C_VEL
LIN {X 0,Y 573.245,Z 362.574,A -85,B 0,C 180,E1 -2117.357,E2 -2117.357} C_VEL
LIN {X 0,Y 573.241,Z 362.578,A -85,B 0,C 180,E1 -2120.393,E2 -2120.393} C_VEL
LIN {X 0,Y 573.249,Z 362.576,A -85,B 0,C 180,E1 -2123.078,E2 -2123.078} C_VEL
LIN {X 0,Y 573.266,Z 362.568,A -85,B 0,C 180,E1 -2125.672,E2 -2125.672} C_VEL
LIN {X 0,Y 573.245,Z 362.577,A -85,B 0,C 180,E1 -2128.185,E2 -2128.185} C_VEL
LIN {X 0,Y 573.263,Z 362.578,A -85,B 0,C 180,E1 -2130.635,E2 -2130.635} C_VEL
LIN {X 0,Y 573.263,Z 362.569,A -85,B 0,C 180,E1 -2133.501,E2 -2133.501} C_VEL
LIN {X 0,Y 573.226,Z 362.579,A -85,B 0,C 180,E1 -2136.135,E2 -2136.135} C_VEL
LIN {X 0,Y 573.255,Z 362.571,A -85,B 0,C 180,E1 -2139.174,E2 -2139.174} C_VEL
LIN {X 0,Y 573.232,Z 362.572,A -85,B 0,C 180,E1 -2141.412,E2 -2141.412} C_VEL
LIN {X 0,Y 573.253,Z 362.572,A -85,B 0,C 180,E1 -2143.622,E2 -2143.622} C_VEL
LIN {X 0,Y 573.231,Z 362.583,A -85,B 0,C 180,E1 -2146.53,E2 -2146.53} C_VEL
LIN {X 0,Y 573.255,Z 362.573,A -85,B 0,C 180,E1 -2148.745,E2 -2148.745} C_VEL
LIN {X 0,Y 573.285,Z 362.566,A -85,B 0,C 180,E1 -2151.541,E2 -2151.541} C_VEL
LIN {X 0,Y 573.287,Z 362.578,A -85,B 0,C 180,E1 -2154.372,E2 -2154.372} C_VEL
LIN {X 0,Y 573.305,Z 362.567,A -85,B 0,C 180,E1 -2157.893,E2 -2157.893} C_VEL
LIN {X 0,Y 573.33,Z 362.565,A -85,B 0,C 180,E1 -2160.703,E2 -2160.703} C_VEL
LIN {X 0,Y 573.235,Z 362.575,A -85,B 0,C 180,E1 -2163.515,E2 -2163.515} C_VEL
LIN {X 0,Y 573.288,Z 362.569,A -85,B 0,C 180,E1 -2165.629,E2 -2165.629} C_VEL
LIN {X 0,Y 573.286,Z 362.571,A -85,B 0,C 180,E1 -2168.46,E2 -2168.46} C_VEL
LIN {X 0,Y 573.266,Z 362.569,A -85,B 0,C 180,E1 -2171.312,E2 -2171.312} C_VEL
LIN {X 0,Y 573.268,Z 362.579,A -85,B 0,C 180,E1 -2174.193,E2 -2174.193} C_VEL
LIN {X 0,Y 573.255,Z 362.57,A -85,B 0,C 180,E1 -2177.112,E2 -2177.112} C_VEL
LIN {X 0,Y 573.252,Z 362.577,A -85,B 0,C 180,E1 -2180.077,E2 -2180.077} C_VEL
LIN {X 0,Y 573.235,Z 362.582,A -85,B 0,C 180,E1 -2182.338,E2 -2182.338} C_VEL
LIN {X 0,Y 573.252,Z 362.571,A -85,B 0,C 180,E1 -2185.411,E2 -2185.411} C_VEL
LIN {X 0,Y 573.26,Z 362.577,A -85,B 0,C 180,E1 -2188.032,E2 -2188.032} C_VEL
LIN {X 0,Y 573.241,Z 362.574,A -85,B 0,C 180,E1 -2190.886,E2 -2190.886} C_VEL
LIN {X 0,Y 573.285,Z 362.568,A -85,B 0,C 180,E1 -2193.529,E2 -2193.529} C_VEL
LIN {X 0,Y 573.258,Z 362.58,A -85,B 0,C 180,E1 -2196.049,E2 -2196.049} C_VEL
LIN {X 0,Y 573.247,Z 362.574,A -85,B 0,C 180,E1 -2198.702,E2 -2198.702} C_VEL
LIN {X 0,Y 573.252,Z 362.575,A -85,B 0,C 180,E1 -2201.596,E2 -2201.596} C_VEL
LIN {X 0,Y 573.238,Z 362.579,A -85,B 0,C 180,E1 -2204.334,E2 -2204.334} C_VEL
LIN {X 0,Y 573.239,Z 362.575,A -85,B 0,C 180,E1 -2207.359,E2 -2207.359} C_VEL
LIN {X 0,Y 573.248,Z 362.577,A -85,B 0,C 180,E1 -2210.394,E2 -2210.394} C_VEL
LIN {X 0,Y 573.256,Z 362.572,A -85,B 0,C 180,E1 -2213.079,E2 -2213.079} C_VEL
LIN {X 0,Y 573.275,Z 362.575,A -85,B 0,C 180,E1 -2215.673,E2 -2215.673} C_VEL
LIN {X 0,Y 573.246,Z 362.58,A -85,B 0,C 180,E1 -2218.186,E2 -2218.186} C_VEL
LIN {X 0,Y 573.27,Z 362.573,A -85,B 0,C 180,E1 -2220.635,E2 -2220.635} C_VEL
LIN {X 0,Y 573.252,Z 362.575,A -85,B 0,C 180,E1 -2223.025,E2 -2223.025} C_VEL
LIN {X 0,Y 573.291,Z 362.782,A -85,B 0,C 180,E1 -2225.118,E2 -2225.118} C_VEL
LIN {X 0,Y 573.848,Z 367.185,A -85,B 0,C 180,E1 -2225.97,E2 -2225.97} C_VEL
LIN {X 0,Y 573.684,Z 383.237,A -85,B 0,C 180,E1 -2228.892,E2 -2228.892} C_VEL
LIN {X 0,Y 573.514,Z 400.404,A -85,B 0,C 180,E1 -2231.976,E2 -2231.976} C_VEL
LIN {X 0,Y 573.343,Z 417.995,A -85,B 0,C 180,E1 -2235.084,E2 -2235.084} C_VEL
LIN {X 0,Y 573.301,Z 424.248,A -85,B 0,C 180,E1 -2236.147,E2 -2236.147} C_VEL
LIN {X 0,Y 573.619,Z 426.345,A -85,B 0,C 180,E1 -2236.218,E2 -2236.218} C_VEL
LIN {X 0,Y 574.071,Z 430.327,A -85,B 0,C 180,E1 -2236.279,E2 -2236.279} C_VEL
LIN {X 0,Y 573.885,Z 530.696,A -85,B 0,C 180,E1 -2237.558,E2 -2237.558} C_VEL
LIN {X 0,Y 573.812,Z 542.636,A -85,B 0,C 180,E1 -2237.826,E2 -2237.826} C_VEL
LIN {X 0,Y 573.7,Z 556.415,A -85,B 0,C 180,E1 -2238.294,E2 -2238.294} C_VEL
LIN {X 0,Y 573.588,Z 568.643,A -85,B 0,C 180,E1 -2238.878,E2 -2238.878} C_VEL
LIN {X 0,Y 573.455,Z 578.849,A -85,B 0,C 180,E1 -2239.497,E2 -2239.497} C_VEL
LIN {X 0,Y 573.354,Z 588.429,A -85,B 0,C 180,E1 -2240.208,E2 -2240.208} C_VEL
LIN {X 0,Y 573.253,Z 597.321,A -85,B 0,C 180,E1 -2241.007,E2 -2241.007} C_VEL
LIN {X 0,Y 573.161,Z 606.964,A -85,B 0,C 180,E1 -2242.071,E2 -2242.071} C_VEL
LIN {X 0,Y 573.07,Z 614.596,A -85,B 0,C 180,E1 -2243.131,E2 -2243.131} C_VEL
LIN {X 0,Y 573.073,Z 619.85,A -85,B 0,C 180,E1 -2244.017,E2 -2244.017} C_VEL
LIN {X 0,Y 572.963,Z 624.919,A -85,B 0,C 180,E1 -2245.075,E2 -2245.075} C_VEL
LIN {X 0,Y 573.014,Z 628.86,A -85,B 0,C 180,E1 -2246.132,E2 -2246.132} C_VEL
LIN {X 0,Y 572.959,Z 631.775,A -85,B 0,C 180,E1 -2247.188,E2 -2247.188} C_VEL
LIN {X 0,Y 572.938,Z 633.209,A -85,B 0,C 180,E1 -2247.891,E2 -2247.891} C_VEL
LIN {X 0,Y 572.94,Z 634.772,A -85,B 0,C 180,E1 -2249.297,E2 -2249.297} C_VEL
LIN {X 0,Y 572.938,Z 635,A -85,B 0,C 180,E1 -2250,E2 -2250} C_VEL
LIN {X 0,Y 572.946,Z 634.18,A -85,B 0,C 180,E1 -2251.406,E2 -2251.406} C_VEL
LIN {X 0,Y 572.938,Z 633.208,A -85,B 0,C 180,E1 -2252.109,E2 -2252.109} C_VEL
LIN {X 0,Y 573.022,Z 629.936,A -85,B 0,C 180,E1 -2253.516,E2 -2253.516} C_VEL
LIN {X 0,Y 573.028,Z 626.337,A -85,B 0,C 180,E1 -2254.573,E2 -2254.573} C_VEL
LIN {X 0,Y 573.068,Z 621.645,A -85,B 0,C 180,E1 -2255.631,E2 -2255.631} C_VEL
LIN {X 0,Y 573.089,Z 616.16,A -85,B 0,C 180,E1 -2256.618,E2 -2256.618} C_VEL
LIN {X 0,Y 573.143,Z 609.656,A -85,B 0,C 180,E1 -2257.575,E2 -2257.575} C_VEL
LIN {X 0,Y 573.207,Z 600.79,A -85,B 0,C 180,E1 -2258.638,E2 -2258.638} C_VEL
LIN {X 0,Y 573.325,Z 590.584,A -85,B 0,C 180,E1 -2259.615,E2 -2259.615} C_VEL
LIN {X 0,Y 573.432,Z 580.153,A -85,B 0,C 180,E1 -2260.415,E2 -2260.415} C_VEL
LIN {X 0,Y 573.57,Z 570.247,A -85,B 0,C 180,E1 -2261.032,E2 -2261.032} C_VEL
LIN {X 0,Y 573.678,Z 559.624,A -85,B 0,C 180,E1 -2261.563,E2 -2261.563} C_VEL
LIN {X 0,Y 573.755,Z 549.113,A -85,B 0,C 180,E1 -2261.974,E2 -2261.974} C_VEL
LIN {X 0,Y 573.861,Z 536.489,A -85,B 0,C 180,E1 -2262.331,E2 -2262.331} C_VEL
LIN {X 0,Y 573.905,Z 521.516,A -85,B 0,C 180,E1 -2262.577,E2 -2262.577} C_VEL
LIN {X 0,Y 573.941,Z 428.304,A -85,B 0,C 180,E1 -2263.749,E2 -2263.749} C_VEL
LIN {X 0,Y 573.339,Z 424.559,A -85,B 0,C 180,E1 -2263.829,E2 -2263.829} C_VEL
LIN {X 0,Y 573.29,Z 422.132,A -85,B 0,C 180,E1 -2264.193,E2 -2264.193} C_VEL
LIN {X 0,Y 573.434,Z 407.771,A -85,B 0,C 180,E1 -2266.717,E2 -2266.717} C_VEL
LIN {X 0,Y 573.58,Z 392.949,A -85,B 0,C 180,E1 -2269.357,E2 -2269.357} C_VEL
LIN {X 0,Y 573.733,Z 376.601,A -85,B 0,C 180,E1 -2272.317,E2 -2272.317} C_VEL
LIN {X 0,Y 573.841,Z 366.156,A -85,B 0,C 180,E1 -2274.223,E2 -2274.223} C_VEL
LIN {X 0,Y 573.271,Z 362.629,A -85,B 0,C 180,E1 -2274.955,E2 -2274.955} C_VEL
LIN {X 0,Y 573.267,Z 362.58,A -85,B 0,C 180,E1 -2278.031,E2 -2278.031} C_VEL
LIN {X 0,Y 573.237,Z 362.576,A -85,B 0,C 180,E1 -2280.883,E2 -2280.883} C_VEL
LIN {X 0,Y 573.265,Z 362.573,A -85,B 0,C 180,E1 -2283.524,E2 -2283.524} C_VEL
LIN {X 0,Y 573.264,Z 362.579,A -85,B 0,C 180,E1 -2286.048,E2 -2286.048} C_VEL
LIN {X 0,Y 573.251,Z 362.574,A -85,B 0,C 180,E1 -2288.701,E2 -2288.701} C_VEL
LIN {X 0,Y 573.254,Z 362.573,A -85,B 0,C 180,E1 -2291.595,E2 -2291.595} C_VEL
LIN {X 0,Y 573.236,Z 362.578,A -85,B 0,C 180,E1 -2294.333,E2 -2294.333} C_VEL
LIN {X 0,Y 573.245,Z 362.575,A -85,B 0,C 180,E1 -2297.358,E2 -2297.358} C_VEL
LIN {X 0,Y 573.248,Z 362.575,A -85,B 0,C 180,E1 -2300.393,E2 -2300.393} C_VEL
LIN {X 0,Y 573.256,Z 362.572,A -85,B 0,C 180,E1 -2303.077,E2 -2303.077} C_VEL
LIN {X 0,Y 573.268,Z 362.576,A -85,B 0,C 180,E1 -2305.671,E2 -2305.671} C_VEL
LIN {X 0,Y 573.25,Z 362.578,A -85,B 0,C 180,E1 -2308.185,E2 -2308.185} C_VEL
LIN {X 0,Y 573.268,Z 362.571,A -85,B 0,C 180,E1 -2310.634,E2 -2310.634} C_VEL
LIN {X 0,Y 573.251,Z 362.57,A -85,B 0,C 180,E1 -2313.024,E2 -2313.024} C_VEL
LIN {X 0,Y 573.274,Z 362.571,A -85,B 0,C 180,E1 -2315.366,E2 -2315.366} C_VEL
LIN {X 0,Y 573.229,Z 362.576,A -85,B 0,C 180,E1 -2318.419,E2 -2318.419} C_VEL
LIN {X 0,Y 573.277,Z 362.566,A -85,B 0,C 180,E1 -2320.728,E2 -2320.728} C_VEL
LIN {X 0,Y 573.257,Z 362.577,A -85,B 0,C 180,E1 -2323.622,E2 -2323.622} C_VEL
LIN {X 0,Y 573.272,Z 362.579,A -85,B 0,C 180,E1 -2325.807,E2 -2325.807} C_VEL
LIN {X 0,Y 573.26,Z 362.569,A -85,B 0,C 180,E1 -2328.745,E2 -2328.745} C_VEL
LIN {X 0,Y 573.288,Z 362.57,A -85,B 0,C 180,E1 -2331.54,E2 -2331.54} C_VEL
LIN {X 0,Y 573.289,Z 362.569,A -85,B 0,C 180,E1 -2334.371,E2 -2334.371} C_VEL
LIN {X 0,Y 573.307,Z 362.57,A -85,B 0,C 180,E1 -2337.892,E2 -2337.892} C_VEL
LIN {X 0,Y 573.332,Z 362.558,A -85,B 0,C 180,E1 -2340.702,E2 -2340.702} C_VEL
LIN {X 0,Y 573.236,Z 362.581,A -85,B 0,C 180,E1 -2343.514,E2 -2343.514} C_VEL
LIN {X 0,Y 573.288,Z 362.578,A -85,B 0,C 180,E1 -2345.628,E2 -2345.628} C_VEL
LIN {X 0,Y 573.287,Z 362.566,A -85,B 0,C 180,E1 -2348.459,E2 -2348.459} C_VEL
LIN {X 0,Y 573.268,Z 362.572,A -85,B 0,C 180,E1 -2351.312,E2 -2351.312} C_VEL
LIN {X 0,Y 573.27,Z 362.572,A -85,B 0,C 180,E1 -2354.193,E2 -2354.193} C_VEL
LIN {X 0,Y 573.255,Z 362.575,A -85,B 0,C 180,E1 -2357.111,E2 -2357.111} C_VEL
LIN {X 0,Y 573.25,Z 362.573,A -85,B 0,C 180,E1 -2360.076,E2 -2360.076} C_VEL
LIN {X 0,Y 573.23,Z 362.579,A -85,B 0,C 180,E1 -2363.099,E2 -2363.099} C_VEL
LIN {X 0,Y 573.247,Z 362.573,A -85,B 0,C 180,E1 -2364.395,E2 -2364.395} C_VEL
LIN {X 0,Y 572.621,Z 362.655,A -85,B 0,C 180,E1 -2364.981,E2 -2364.981} C_VEL
LIN {X 0,Y 569.783,Z 363.012,A -85,B 0,C 180,E1 -2365.933,E2 -2365.933} C_VEL
LIN {X 0,Y 567.355,Z 363.316,A -85,B 0,C 180,E1 -2366.699,E2 -2366.699} C_VEL
LIN {X 0,Y 566.302,Z 363.444,A -85,B 0,C 180,E1 -2367.29,E2 -2367.29} C_VEL
LIN {X 0,Y 566.213,Z 363.453,A -85,B 0,C 180,E1 -2367.49,E2 -2367.49} C_VEL
LIN {X 0,Y 566.184,Z 363.453,A -85,B 0,C 180,E1 -2370.592,E2 -2370.592} C_VEL
LIN {X 0,Y 566.225,Z 363.453,A -85,B 0,C 180,E1 -2373.101,E2 -2373.101} C_VEL
LIN {X 0,Y 566.208,Z 363.455,A -85,B 0,C 180,E1 -2375.688,E2 -2375.688} C_VEL
LIN {X 0,Y 566.211,Z 363.45,A -85,B 0,C 180,E1 -2378.559,E2 -2378.559} C_VEL
LIN {X 0,Y 566.208,Z 363.454,A -85,B 0,C 180,E1 -2381.136,E2 -2381.136} C_VEL
LIN {X 0,Y 566.196,Z 363.452,A -85,B 0,C 180,E1 -2384.035,E2 -2384.035} C_VEL
LIN {X 0,Y 566.197,Z 363.454,A -85,B 0,C 180,E1 -2387.083,E2 -2387.083} C_VEL
LIN {X 0,Y 566.223,Z 363.449,A -85,B 0,C 180,E1 -2389.803,E2 -2389.803} C_VEL
LIN {X 0,Y 566.195,Z 363.453,A -85,B 0,C 180,E1 -2392.599,E2 -2392.599} C_VEL
LIN {X 0,Y 566.219,Z 363.454,A -85,B 0,C 180,E1 -2395.183,E2 -2395.183} C_VEL
LIN {X 0,Y 566.231,Z 363.45,A -85,B 0,C 180,E1 -2397.744,E2 -2397.744} C_VEL
LIN {X 0,Y 566.225,Z 363.446,A -85,B 0,C 180,E1 -2400.323,E2 -2400.323} C_VEL
LIN {X 0,Y 566.216,Z 363.452,A -85,B 0,C 180,E1 -2402.661,E2 -2402.661} C_VEL
LIN {X 0,Y 566.233,Z 363.455,A -85,B 0,C 180,E1 -2405.039,E2 -2405.039} C_VEL
LIN {X 0,Y 566.191,Z 363.453,A -85,B 0,C 180,E1 -2408.137,E2 -2408.137} C_VEL
LIN {X 0,Y 566.233,Z 363.45,A -85,B 0,C 180,E1 -2410.612,E2 -2410.612} C_VEL
LIN {X 0,Y 566.213,Z 363.456,A -85,B 0,C 180,E1 -2413.412,E2 -2413.412} C_VEL
LIN {X 0,Y 566.195,Z 363.453,A -85,B 0,C 180,E1 -2416.359,E2 -2416.359} C_VEL
LIN {X 0,Y 566.232,Z 363.452,A -85,B 0,C 180,E1 -2418.675,E2 -2418.675} C_VEL
LIN {X 0,Y 566.225,Z 363.453,A -85,B 0,C 180,E1 -2421.434,E2 -2421.434} C_VEL
LIN {X 0,Y 566.266,Z 363.445,A -85,B 0,C 180,E1 -2424.302,E2 -2424.302} C_VEL
LIN {X 0,Y 566.283,Z 363.442,A -85,B 0,C 180,E1 -2427.866,E2 -2427.866} C_VEL
LIN {X 0,Y 566.299,Z 363.445,A -85,B 0,C 180,E1 -2430.711,E2 -2430.711} C_VEL
LIN {X 0,Y 566.268,Z 363.451,A -85,B 0,C 180,E1 -2432.845,E2 -2432.845} C_VEL
LIN {X 0,Y 566.265,Z 363.445,A -85,B 0,C 180,E1 -2435.698,E2 -2435.698} C_VEL
LIN {X 0,Y 566.23,Z 363.453,A -85,B 0,C 180,E1 -2438.565,E2 -2438.565} C_VEL
LIN {X 0,Y 566.238,Z 363.45,A -85,B 0,C 180,E1 -2441.454,E2 -2441.454} C_VEL
LIN {X 0,Y 566.231,Z 363.452,A -85,B 0,C 180,E1 -2444.507,E2 -2444.507} C_VEL
LIN {X 0,Y 566.2,Z 363.455,A -85,B 0,C 180,E1 -2447.331,E2 -2447.331} C_VEL
LIN {X 0,Y 566.21,Z 363.453,A -85,B 0,C 180,E1 -2450.337,E2 -2450.337} C_VEL
LIN {X 0,Y 566.185,Z 363.456,A -85,B 0,C 180,E1 -2453.404,E2 -2453.404} C_VEL
LIN {X 0,Y 566.22,Z 363.449,A -85,B 0,C 180,E1 -2455.748,E2 -2455.748} C_VEL
LIN {X 0,Y 566.202,Z 363.453,A -85,B 0,C 180,E1 -2458.203,E2 -2458.203} C_VEL
LIN {X 0,Y 566.189,Z 363.457,A -85,B 0,C 180,E1 -2460.592,E2 -2460.592} C_VEL
LIN {X 0,Y 566.223,Z 363.451,A -85,B 0,C 180,E1 -2463.101,E2 -2463.101} C_VEL
LIN {X 0,Y 566.208,Z 363.448,A -85,B 0,C 180,E1 -2465.688,E2 -2465.688} C_VEL
LIN {X 0,Y 566.211,Z 363.457,A -85,B 0,C 180,E1 -2468.559,E2 -2468.559} C_VEL
LIN {X 0,Y 566.202,Z 363.447,A -85,B 0,C 180,E1 -2471.136,E2 -2471.136} C_VEL
LIN {X 0,Y 566.193,Z 363.45,A -85,B 0,C 180,E1 -2474.035,E2 -2474.035} C_VEL
LIN {X 0,Y 566.203,Z 363.454,A -85,B 0,C 180,E1 -2477.082,E2 -2477.082} C_VEL
LIN {X 0,Y 566.22,Z 363.447,A -85,B 0,C 180,E1 -2479.803,E2 -2479.803} C_VEL
LIN {X 0,Y 566.192,Z 363.462,A -85,B 0,C 180,E1 -2482.599,E2 -2482.599} C_VEL
LIN {X 0,Y 566.213,Z 363.448,A -85,B 0,C 180,E1 -2485.183,E2 -2485.183} C_VEL
LIN {X 0,Y 566.23,Z 363.447,A -85,B 0,C 180,E1 -2487.744,E2 -2487.744} C_VEL
LIN {X 0,Y 566.221,Z 363.454,A -85,B 0,C 180,E1 -2490.323,E2 -2490.323} C_VEL
LIN {X 0,Y 566.227,Z 363.446,A -85,B 0,C 180,E1 -2493.335,E2 -2493.335} C_VEL
LIN {X 0,Y 566.192,Z 363.453,A -85,B 0,C 180,E1 -2495.82,E2 -2495.82} C_VEL
LIN {X 0,Y 566.21,Z 363.451,A -85,B 0,C 180,E1 -2498.903,E2 -2498.903} C_VEL
LIN {X 0,Y 566.206,Z 363.448,A -85,B 0,C 180,E1 -2501.173,E2 -2501.173} C_VEL
LIN {X 0,Y 566.215,Z 363.448,A -85,B 0,C 180,E1 -2503.413,E2 -2503.413} C_VEL
LIN {X 0,Y 566.194,Z 363.461,A -85,B 0,C 180,E1 -2506.359,E2 -2506.359} C_VEL
LIN {X 0,Y 566.227,Z 363.449,A -85,B 0,C 180,E1 -2508.675,E2 -2508.675} C_VEL
LIN {X 0,Y 566.228,Z 363.445,A -85,B 0,C 180,E1 -2511.435,E2 -2511.435} C_VEL
LIN {X 0,Y 566.255,Z 363.452,A -85,B 0,C 180,E1 -2514.302,E2 -2514.302} C_VEL
LIN {X 0,Y 566.276,Z 363.442,A -85,B 0,C 180,E1 -2517.867,E2 -2517.867} C_VEL
LIN {X 0,Y 566.3,Z 363.44,A -85,B 0,C 180,E1 -2520.711,E2 -2520.711} C_VEL
LIN {X 0,Y 566.272,Z 363.444,A -85,B 0,C 180,E1 -2522.846,E2 -2522.846} C_VEL
LIN {X 0,Y 566.256,Z 363.445,A -85,B 0,C 180,E1 -2525.699,E2 -2525.699} C_VEL
LIN {X 0,Y 566.229,Z 363.447,A -85,B 0,C 180,E1 -2528.566,E2 -2528.566} C_VEL
LIN {X 0,Y 566.236,Z 363.444,A -85,B 0,C 180,E1 -2531.455,E2 -2531.455} C_VEL
LIN {X 0,Y 566.229,Z 363.452,A -85,B 0,C 180,E1 -2534.507,E2 -2534.507} C_VEL
LIN {X 0,Y 566.2,Z 363.448,A -85,B 0,C 180,E1 -2537.332,E2 -2537.332} C_VEL
LIN {X 0,Y 566.215,Z 363.456,A -85,B 0,C 180,E1 -2540.337,E2 -2540.337} C_VEL
LIN {X 0,Y 566.186,Z 363.453,A -85,B 0,C 180,E1 -2543.404,E2 -2543.404} C_VEL
LIN {X 0,Y 566.221,Z 363.45,A -85,B 0,C 180,E1 -2545.749,E2 -2545.749} C_VEL
LIN {X 0,Y 566.203,Z 363.459,A -85,B 0,C 180,E1 -2548.204,E2 -2548.204} C_VEL
LIN {X 0,Y 566.191,Z 363.455,A -85,B 0,C 180,E1 -2550.593,E2 -2550.593} C_VEL
LIN {X 0,Y 566.226,Z 363.446,A -85,B 0,C 180,E1 -2553.102,E2 -2553.102} C_VEL
LIN {X 0,Y 566.209,Z 363.452,A -85,B 0,C 180,E1 -2555.689,E2 -2555.689} C_VEL
LIN {X 0,Y 566.214,Z 363.451,A -85,B 0,C 180,E1 -2558.56,E2 -2558.56} C_VEL
LIN {X 0,Y 566.21,Z 363.449,A -85,B 0,C 180,E1 -2561.137,E2 -2561.137} C_VEL
LIN {X 0,Y 566.199,Z 363.46,A -85,B 0,C 180,E1 -2564.036,E2 -2564.036} C_VEL
LIN {X 0,Y 566.2,Z 363.451,A -85,B 0,C 180,E1 -2567.083,E2 -2567.083} C_VEL
LIN {X 0,Y 566.227,Z 363.451,A -85,B 0,C 180,E1 -2569.803,E2 -2569.803} C_VEL
LIN {X 0,Y 566.199,Z 363.452,A -85,B 0,C 180,E1 -2572.6,E2 -2572.6} C_VEL
LIN {X 0,Y 566.222,Z 363.449,A -85,B 0,C 180,E1 -2575.184,E2 -2575.184} C_VEL
LIN {X 0,Y 566.233,Z 363.453,A -85,B 0,C 180,E1 -2577.744,E2 -2577.744} C_VEL
LIN {X 0,Y 566.229,Z 363.453,A -85,B 0,C 180,E1 -2580.324,E2 -2580.324} C_VEL
LIN {X 0,Y 566.22,Z 363.452,A -85,B 0,C 180,E1 -2582.662,E2 -2582.662} C_VEL
LIN {X 0,Y 566.254,Z 363.62,A -85,B 0,C 180,E1 -2584.963,E2 -2584.963} C_VEL
LIN {X 0,Y 566.901,Z 369.164,A -85,B 0,C 180,E1 -2586.046,E2 -2586.046} C_VEL
LIN {X 0,Y 566.687,Z 384.862,A -85,B 0,C 180,E1 -2588.921,E2 -2588.921} C_VEL
LIN {X 0,Y 566.509,Z 400.404,A -85,B 0,C 180,E1 -2591.745,E2 -2591.745} C_VEL
LIN {X 0,Y 566.32,Z 416.961,A -85,B 0,C 180,E1 -2594.71,E2 -2594.71} C_VEL
LIN {X 0,Y 566.281,Z 424.255,A -85,B 0,C 180,E1 -2595.972,E2 -2595.972} C_VEL
LIN {X 0,Y 566.609,Z 426.456,A -85,B 0,C 180,E1 -2596.045,E2 -2596.045} C_VEL
LIN {X 0,Y 567.188,Z 432.116,A -85,B 0,C 180,E1 -2596.132,E2 -2596.132} C_VEL
LIN {X 0,Y 566.971,Z 530.641,A -85,B 0,C 180,E1 -2597.404,E2 -2597.404} C_VEL
LIN {X 0,Y 566.866,Z 542.601,A -85,B 0,C 180,E1 -2597.674,E2 -2597.674} C_VEL
LIN {X 0,Y 566.745,Z 556.421,A -85,B 0,C 180,E1 -2598.149,E2 -2598.149} C_VEL
LIN {X 0,Y 566.628,Z 568.042,A -85,B 0,C 180,E1 -2598.707,E2 -2598.707} C_VEL
LIN {X 0,Y 566.468,Z 578.834,A -85,B 0,C 180,E1 -2599.365,E2 -2599.365} C_VEL
LIN {X 0,Y 566.309,Z 588.415,A -85,B 0,C 180,E1 -2600.085,E2 -2600.085} C_VEL
LIN {X 0,Y 566.228,Z 597.309,A -85,B 0,C 180,E1 -2600.895,E2 -2600.895} C_VEL
LIN {X 0,Y 566.112,Z 606.964,A -85,B 0,C 180,E1 -2601.972,E2 -2601.972} C_VEL
LIN {X 0,Y 566.008,Z 614.721,A -85,B 0,C 180,E1 -2603.065,E2 -2603.065} C_VEL
LIN {X 0,Y 565.989,Z 619.846,A -85,B 0,C 180,E1 -2603.942,E2 -2603.942} C_VEL
LIN {X 0,Y 565.878,Z 624.913,A -85,B 0,C 180,E1 -2605.013,E2 -2605.013} C_VEL
LIN {X 0,Y 565.926,Z 628.853,A -85,B 0,C 180,E1 -2606.084,E2 -2606.084} C_VEL
LIN {X 0,Y 565.878,Z 631.767,A -85,B 0,C 180,E1 -2607.153,E2 -2607.153} C_VEL
LIN {X 0,Y 565.839,Z 633.21,A -85,B 0,C 180,E1 -2607.865,E2 -2607.865} C_VEL
LIN {X 0,Y 565.841,Z 634.764,A -85,B 0,C 180,E1 -2609.289,E2 -2609.289} C_VEL
LIN {X 0,Y 565.839,Z 635,A -85,B 0,C 180,E1 -2610,E2 -2610} C_VEL
LIN {X 0,Y 565.846,Z 634.173,A -85,B 0,C 180,E1 -2611.424,E2 -2611.424} C_VEL
LIN {X 0,Y 565.839,Z 633.209,A -85,B 0,C 180,E1 -2612.136,E2 -2612.136} C_VEL
LIN {X 0,Y 565.927,Z 629.932,A -85,B 0,C 180,E1 -2613.56,E2 -2613.56} C_VEL
LIN {X 0,Y 565.933,Z 626.33,A -85,B 0,C 180,E1 -2614.63,E2 -2614.63} C_VEL
LIN {X 0,Y 565.998,Z 621.637,A -85,B 0,C 180,E1 -2615.701,E2 -2615.701} C_VEL
LIN {X 0,Y 566.017,Z 615.104,A -85,B 0,C 180,E1 -2616.873,E2 -2616.873} C_VEL
LIN {X 0,Y 566.113,Z 606.961,A -85,B 0,C 180,E1 -2618.028,E2 -2618.028} C_VEL
LIN {X 0,Y 566.228,Z 597.304,A -85,B 0,C 180,E1 -2619.106,E2 -2619.106} C_VEL
LIN {X 0,Y 566.31,Z 588.41,A -85,B 0,C 180,E1 -2619.915,E2 -2619.915} C_VEL
LIN {X 0,Y 566.469,Z 578.828,A -85,B 0,C 180,E1 -2620.635,E2 -2620.635} C_VEL
LIN {X 0,Y 566.615,Z 568.165,A -85,B 0,C 180,E1 -2621.287,E2 -2621.287} C_VEL
LIN {X 0,Y 566.759,Z 555.288,A -85,B 0,C 180,E1 -2621.897,E2 -2621.897} C_VEL
LIN {X 0,Y 566.867,Z 542.585,A -85,B 0,C 180,E1 -2622.326,E2 -2622.326} C_VEL
LIN {X 0,Y 566.959,Z 531.937,A -85,B 0,C 180,E1 -2622.574,E2 -2622.574} C_VEL
LIN {X 0,Y 567.075,Z 500.052,A -85,B 0,C 180,E1 -2623.004,E2 -2623.004} C_VEL
LIN {X 0,Y 567.062,Z 429.2,A -85,B 0,C 180,E1 -2623.908,E2 -2623.908} C_VEL
LIN {X 0,Y 566.294,Z 424.569,A -85,B 0,C 180,E1 -2624.005,E2 -2624.005} C_VEL
LIN {X 0,Y 566.26,Z 422.132,A -85,B 0,C 180,E1 -2624.373,E2 -2624.373} C_VEL
LIN {X 0,Y 566.436,Z 405.575,A -85,B 0,C 180,E1 -2627.324,E2 -2627.324} C_VEL
